// TIA Portal project "Shubra" (V16)

(* hardware
DEVICE "S7-1200 station_1"  S7-1200 Station
   slot 0: "Rack_0"  S7-1200 Rack  Rack  V1.0
   slot 1: "PLC_1"  CPU 1214C DC/DC/DC  6ES7 214-1AG40-0XB0  V4.4
   slot 2: "AI 8x13BIT_1"  6ES7 231-4HF32-0XB0  V2.1
DEVICE "PC-System_1"  SIMATIC PC station
   slot 0: "SIMATIC PC station"  Rail  SIMATIC PC-Station  V1.0
      slot 125: "Stationmanager"  Station_Manager  V6.0.4
   slot 1: "HMI_RT_1"  WinCC RT Advanced  6AV2 104-0xxxx-xxxx  16.0.0.0
      slot 33792: "Computer interface"  Host interface
   slot 2: "IE general_1"  IE General  IE_CP  V8.2.0
*)

// ===== PLC "PLC_1"  CPU 1214C DC/DC/DC =====

VAR_GLOBAL   // PLC tag table "Default tag table"
   "Tag_1" AT %IW112 : Int;
   "Tag_4" AT %IW114 : Int;
   "Tag_7" AT %IW116 : Int;
   "Tag_10" AT %IW118 : Int;
   "Tag_14" AT %IW120 : Int;
   "Tag_18" AT %IW122 : Int;
   "Tag_28" AT %IW124 : Int;
   "Tag_31" AT %IW126 : Int;
   "Tag_25" AT %I0.1 : Bool;
   "Tag_26" AT %I0.2 : Bool;
   "Tag_38" AT %I0.3 : Bool;
   "Axis_1_Pulse" AT %Q0.0 : Bool;
   "Axis_1_Direction" AT %Q0.1 : Bool;
   "Tag_17" AT %Q0.2 : Bool;
   "Axis_2_Pulse" AT %Q0.3 : Bool;
   "Axis_2_Direction" AT %Q0.4 : Bool;
   "Tag_22" AT %Q0.5 : Bool;
   "pump_run" AT %Q0.6 : Bool;
   "Tag_37" AT %QW128 : Word;
   "Tag_2" AT %MD40 : Real;
   "Suction_press" AT %MD44 : Real;
   "Tag_5" AT %MD48 : Real;
   "Discharge_Press" AT %MD52 : Real;
   "Tag_8" AT %MD56 : Real;
   "P3" AT %MD60 : Real;
   "Tag_12" AT %MD64 : Real;
   "P4" AT %MD68 : Real;
   "Tag_15" AT %MD72 : Real;
   "Temperature" AT %MD76 : Real;
   "Tag_20" AT %MD80 : Real;
   "Torque" AT %MD84 : Real;
   "Tag_29" AT %MD88 : Real;
   "RPM" AT %MD92 : Real;
   "Tag_32" AT %MD96 : Real;
   "vibration" AT %MD100 : Real;
   "Tag_11" AT %M20.0 : Bool;
   "compare" AT %MD104 : Real;
   "Tag_9" AT %M20.1 : Bool;
   "Tag_19" AT %M20.2 : Bool;
   "Tag_21" AT %M20.3 : Bool;
   "Tag_23" AT %M21.0 : Bool;
   "Tag_24" AT %M21.1 : Bool;
   "distance_1" AT %MD108 : Real;
   "Tag_35" AT %MD120 : Real;
   "Tag_36" AT %MD124 : DWord;
   "p3-p4" AT %MD128 : Real;
   "p3-p4_power5" AT %MD132 : Real;
   "p3-p4_power4" AT %MD136 : Real;
   "p3-p4_power3" AT %MD140 : Real;
   "p3-p4_power2" AT %MD144 : Real;
   "Q" AT %MD148 : Real;
   "VS" AT %MD152 : Real;
   "Vd" AT %MD156 : Real;
   "Vs2" AT %MD160 : Real;
   "Vd2" AT %MD164 : Real;
   "H" AT %MD168 : Real;
   "Shaft_power" AT %MD172 : Real;
   "Referance_motor_speed" AT %MD176 : Real;
   "QARS" AT %MD180 : Real;
   "Ref_speed_2" AT %MD184 : Real;
   "Ref_speed_3" AT %MD188 : Real;
   "motor_speed_2" AT %MD192 : Real;
   "motor_speed_3" AT %MD196 : Real;
   "H_ARS" AT %MD200 : Real;
   "SP_ARS" AT %MD204 : Real;
   "Efficiency" AT %MD208 : Real;
   "Npsh" AT %MD212 : Real;
   "Count_up" AT %M30.0 : Bool;
   "Tag_3" AT %M31.0 : Bool;
   "count_down" AT %M30.1 : Bool;
   "Tag_13" AT %M31.1 : Bool;
   "counter_reset" AT %M30.2 : Bool;
   "Tag_16" AT %MW36 : Int;
   "Raw1" AT %M30.3 : Bool;
   "raw2" AT %M30.4 : Bool;
   "raw3" AT %M30.5 : Bool;
   "raw4" AT %M30.6 : Bool;
   "raw5" AT %M30.7 : Bool;
   "raw6" AT %M31.4 : Bool;
   "record" AT %M31.5 : Bool;
   "stepp1_enab" AT %M31.6 : Bool;
   "stepp1_start" AT %M31.7 : Bool;
   "stepp1_distance" AT %MD216 : Real;
   "Tag_27" AT %M32.1 : Bool;
   "start_motor" AT %M32.2 : Bool;
   "clear All" AT %M32.3 : Bool;
   "open_close" AT %M32.4 : Bool;
   "stepp1_home" AT %M32.5 : Bool;
   "stepp2_home" AT %M32.6 : Bool;
   "stepp2_enab" AT %M32.7 : Bool;
   "stepp2_excut" AT %M33.0 : Bool;
   "stepp2_distance" AT %MD220 : Real;
   "Stepp1_dist_scale" AT %MD224 : Real;
   "Stepp2_dist_scale" AT %MD228 : Real;
   "configuration" AT %MW232 : WChar;
   "date" AT %MW234 : Date;
   "time" AT %MD236 : Time_Of_Day;
   "time_1" AT %MD240 : Time_Of_Day;
   "deviation" AT %MD244 : Real;
   "raw7" AT %M33.1 : Bool;
   "raw8" AT %M33.2 : Bool;
   "raw9" AT %M33.3 : Bool;
   "raw10" AT %M33.4 : Bool;
   "raw11" AT %M33.5 : Bool;
   "raw12" AT %M33.6 : Bool;
   "record1" AT %M33.7 : Bool;
   "Tag_6" AT %MD112 : Real;
END_VAR

DATA_BLOCK "P1P2"   // DB3
{ S7_Optimized_Access := 'TRUE' }
VERSION : 0.1
   VAR
      Pressurep1p2 : Array[0..23] of Real;
   END_VAR
BEGIN
END_DATA_BLOCK

DATA_BLOCK "P3P4"   // DB4
{ S7_Optimized_Access := 'TRUE' }
VERSION : 0.1
   VAR
      Pressure34 : Array[0..23] of Real;
   END_VAR
BEGIN
END_DATA_BLOCK

DATA_BLOCK "TS"   // DB5
{ S7_Optimized_Access := 'TRUE' }
VERSION : 0.1
   VAR
      TS : Array[0..23] of Real;
   END_VAR
BEGIN
END_DATA_BLOCK

DATA_BLOCK "Vib"   // DB6
{ S7_Optimized_Access := 'TRUE' }
VERSION : 0.1
   VAR
      vibration : Array[0..11] of Real;
   END_VAR
BEGIN
END_DATA_BLOCK

DATA_BLOCK "VSVD"   // DB7
{ S7_Optimized_Access := 'TRUE' }
VERSION : 0.1
   VAR
      VsVd : Array[0..23] of Real;
   END_VAR
BEGIN
END_DATA_BLOCK

DATA_BLOCK "QH"   // DB8
{ S7_Optimized_Access := 'TRUE' }
VERSION : 0.1
   VAR
      QH : Array[0..23] of Real;
   END_VAR
BEGIN
END_DATA_BLOCK

DATA_BLOCK "shftP.Pars"   // DB9
{ S7_Optimized_Access := 'TRUE' }
VERSION : 0.1
   VAR
      shaftP : Array[0..23] of Real;
   END_VAR
BEGIN
END_DATA_BLOCK

DATA_BLOCK "QarsHars"   // DB10
{ S7_Optimized_Access := 'TRUE' }
VERSION : 0.1
   VAR
      QarsHars : Array[0..23] of Real;
   END_VAR
BEGIN
END_DATA_BLOCK

DATA_BLOCK "EFF.NPSH"   // DB11
{ S7_Optimized_Access := 'TRUE' }
VERSION : 0.1
   VAR
      "EFF.NPSH" : Array[0..23] of Real;
   END_VAR
BEGIN
END_DATA_BLOCK

DATA_BLOCK "deviation_1"   // DB19
{ S7_Optimized_Access := 'TRUE' }
VERSION : 0.1
   VAR
      deviation : Real;
      deviation_1 : Real;
      deviation_2 : Real;
      deviation_3 : Real;
      deviation_4 : Real;
      deviation_5 : Real;
      deviation_0 : Real;
   END_VAR
BEGIN
END_DATA_BLOCK

// folder: System blocks/Program resources

DATA_BLOCK "IEC_Counter_0_DB"   // DB12
{ S7_Optimized_Access := 'TRUE' }
AUTHOR : Simatic
FAMILY : IEC
NAME : CNTR
VERSION : 1.0
// stored: InstanceOfName IEC_COUNTER
"IEC_COUNTER"
BEGIN
END_DATA_BLOCK

// folder: (top level)

DATA_BLOCK "Axis_1"   // DB1, Motion_DB
{ S7_Optimized_Access := 'TRUE' }
AUTHOR : SIMATIC
FAMILY : BasicMC
NAME : TO_PosAx
VERSION : 7.0
// stored: InstanceOfName TO_PositioningAxis
"TO_PositioningAxis"
BEGIN
   // Axis.OnlinePtoModeCU = 16#0000_0002
   // Axis.DirectionOutputEnabledCU = TRUE
   // Axis.SelectedChannel2EnumCU = %Q0.1
   // Axis.SelectedChannel1EnumCU = %Q0.0
   // Pulse.MinDeltaDeltaFrequencyCU = 0.004
   // Pulse.MaxDeltaDeltaFrequencyCU = 1.0E+10
   // Pulse.MinDeltaFrequencyCU = 0.005
   // Pulse.MaxDeltaFrequencyCU = 9.5E+9
   // Pulse.MinFrequencyCU = 1.0
   // Pulse.MaxFrequencyCU = 100000.0
   // Pulse.OutputSourceCU = 16#0000_0000
   // Axis.SelectPTO = 0
END_DATA_BLOCK

DATA_BLOCK "Axis_2"   // DB2, Motion_DB
{ S7_Optimized_Access := 'TRUE' }
AUTHOR : SIMATIC
FAMILY : BasicMC
NAME : TO_PosAx
VERSION : 7.0
// stored: InstanceOfName TO_PositioningAxis
"TO_PositioningAxis"
BEGIN
   // Axis.OnlinePtoModeCU = 16#0000_0002
   // Axis.DirectionOutputEnabledCU = TRUE
   // Axis.SelectedChannel2EnumCU = %Q0.4
   // Axis.SelectedChannel1EnumCU = %Q0.3
   // Pulse.MinDeltaDeltaFrequencyCU = 0.004
   // Pulse.MaxDeltaDeltaFrequencyCU = 1.0E+10
   // Pulse.MinDeltaFrequencyCU = 0.005
   // Pulse.MaxDeltaFrequencyCU = 9.5E+9
   // Pulse.MinFrequencyCU = 1.0
   // Pulse.MaxFrequencyCU = 100000.0
   // Pulse.OutputSourceCU = 16#0000_0000
   // Axis.SelectPTO = 1
   // Axis.OnlinePtoIndexCU = 1
END_DATA_BLOCK

FUNCTION "Analog input" : Void   // FC1, LAD
{ S7_Optimized_Access := 'TRUE' }
VERSION : 0.1
BEGIN

REGION Network 1: suction pressure
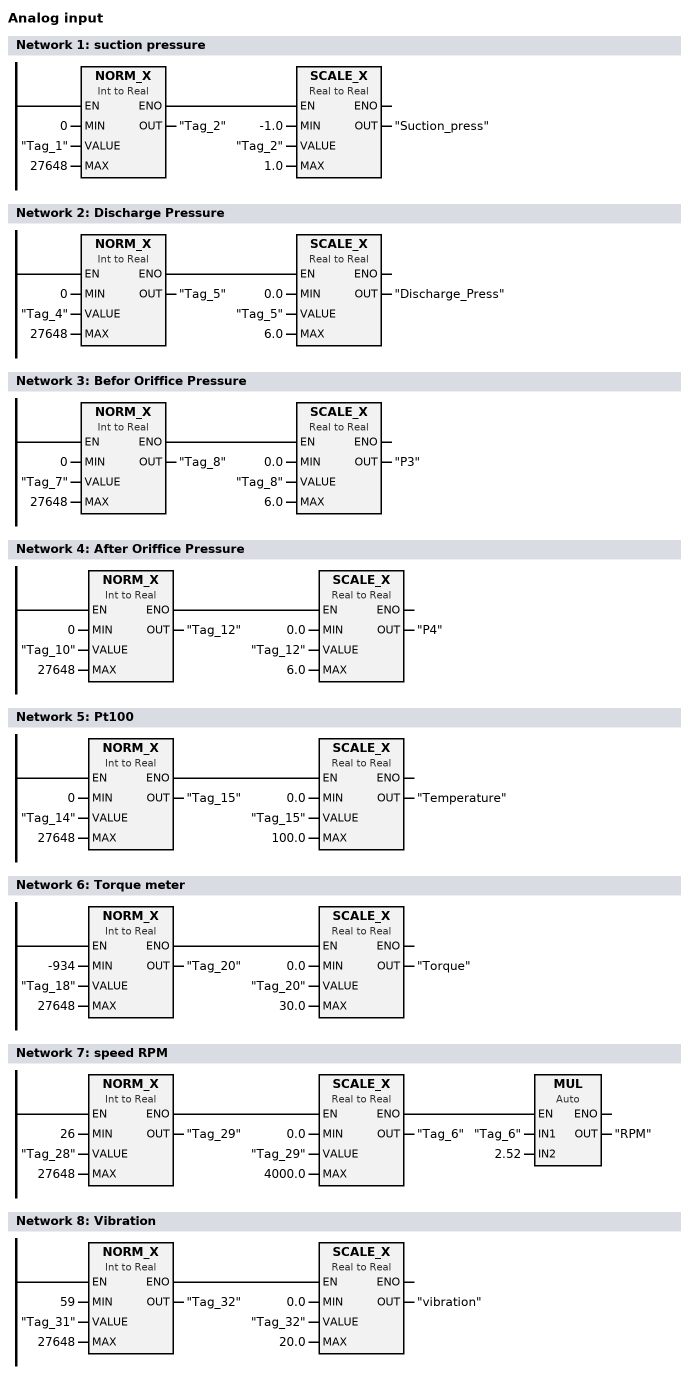
   RUNG wire#powerrail
      { S7_Templates := "[SrcType := Int, DestType := Real]" } Normalize(min := 0, value := "Tag_1", max := 27648, out => "Tag_2")
      { S7_Templates := "[SrcType := Real, DestType := Real]" } Scale(min := -1.0, value := "Tag_2", max := 1.0, out => "Suction_press")
   END_RUNG
   // the same network as SCL:
   "Tag_2" := NORM_X(MIN := 0, VALUE := "Tag_1", MAX := 27648);
   "Suction_press" := SCALE_X(MIN := -1.0, VALUE := "Tag_2", MAX := 1.0);
END_REGION

REGION Network 2: Discharge Pressure
   RUNG wire#powerrail
      { S7_Templates := "[SrcType := Int, DestType := Real]" } Normalize(min := 0, value := "Tag_4", max := 27648, out => "Tag_5")
      { S7_Templates := "[SrcType := Real, DestType := Real]" } Scale(min := 0.0, value := "Tag_5", max := 6.0, out => "Discharge_Press")
   END_RUNG
   // the same network as SCL:
   "Tag_5" := NORM_X(MIN := 0, VALUE := "Tag_4", MAX := 27648);
   "Discharge_Press" := SCALE_X(MIN := 0.0, VALUE := "Tag_5", MAX := 6.0);
END_REGION

REGION Network 3: Befor Oriffice Pressure
   RUNG wire#powerrail
      { S7_Templates := "[SrcType := Int, DestType := Real]" } Normalize(min := 0, value := "Tag_7", max := 27648, out => "Tag_8")
      { S7_Templates := "[SrcType := Real, DestType := Real]" } Scale(min := 0.0, value := "Tag_8", max := 6.0, out => "P3")
   END_RUNG
   // the same network as SCL:
   "Tag_8" := NORM_X(MIN := 0, VALUE := "Tag_7", MAX := 27648);
   "P3" := SCALE_X(MIN := 0.0, VALUE := "Tag_8", MAX := 6.0);
END_REGION

REGION Network 4: After Oriffice Pressure
   RUNG wire#powerrail
      { S7_Templates := "[SrcType := Int, DestType := Real]" } Normalize(min := 0, value := "Tag_10", max := 27648, out => "Tag_12")
      { S7_Templates := "[SrcType := Real, DestType := Real]" } Scale(min := 0.0, value := "Tag_12", max := 6.0, out => "P4")
   END_RUNG
   // the same network as SCL:
   "Tag_12" := NORM_X(MIN := 0, VALUE := "Tag_10", MAX := 27648);
   "P4" := SCALE_X(MIN := 0.0, VALUE := "Tag_12", MAX := 6.0);
END_REGION

REGION Network 5: Pt100
   RUNG wire#powerrail
      { S7_Templates := "[SrcType := Int, DestType := Real]" } Normalize(min := 0, value := "Tag_14", max := 27648, out => "Tag_15")
      { S7_Templates := "[SrcType := Real, DestType := Real]" } Scale(min := 0.0, value := "Tag_15", max := 100.0, out => "Temperature")
   END_RUNG
   // the same network as SCL:
   "Tag_15" := NORM_X(MIN := 0, VALUE := "Tag_14", MAX := 27648);
   "Temperature" := SCALE_X(MIN := 0.0, VALUE := "Tag_15", MAX := 100.0);
END_REGION

REGION Network 6: Torque meter
   RUNG wire#powerrail
      { S7_Templates := "[SrcType := Int, DestType := Real]" } Normalize(min := -934, value := "Tag_18", max := 27648, out => "Tag_20")
      { S7_Templates := "[SrcType := Real, DestType := Real]" } Scale(min := 0.0, value := "Tag_20", max := 30.0, out => "Torque")
   END_RUNG
   // the same network as SCL:
   "Tag_20" := NORM_X(MIN := -934, VALUE := "Tag_18", MAX := 27648);
   "Torque" := SCALE_X(MIN := 0.0, VALUE := "Tag_20", MAX := 30.0);
END_REGION

REGION Network 7: speed RPM
   RUNG wire#powerrail
      { S7_Templates := "[SrcType := Int, DestType := Real]" } Normalize(min := 26, value := "Tag_28", max := 27648, out => "Tag_29")
      { S7_Templates := "[SrcType := Real, DestType := Real]" } Scale(min := 0.0, value := "Tag_29", max := 4000.0, out => "Tag_6")
      Mul(in1 := "Tag_6", in2 := 2.52, out => "RPM")
   END_RUNG
   // the same network as SCL:
   "Tag_29" := NORM_X(MIN := 26, VALUE := "Tag_28", MAX := 27648);
   "Tag_6" := SCALE_X(MIN := 0.0, VALUE := "Tag_29", MAX := 4000.0);
   "RPM" := "Tag_6" * 2.52;
END_REGION

REGION Network 8: Vibration
   RUNG wire#powerrail
      { S7_Templates := "[SrcType := Int, DestType := Real]" } Normalize(min := 59, value := "Tag_31", max := 27648, out => "Tag_32")
      { S7_Templates := "[SrcType := Real, DestType := Real]" } Scale(min := 0.0, value := "Tag_32", max := 20.0, out => "vibration")
   END_RUNG
   // the same network as SCL:
   "Tag_32" := NORM_X(MIN := 59, VALUE := "Tag_31", MAX := 27648);
   "vibration" := SCALE_X(MIN := 0.0, VALUE := "Tag_32", MAX := 20.0);
END_REGION
END_FUNCTION

FUNCTION "clear_2" : Void   // FC2, LAD
{ S7_Optimized_Access := 'TRUE' }
VERSION : 0.1
BEGIN

REGION Network 2
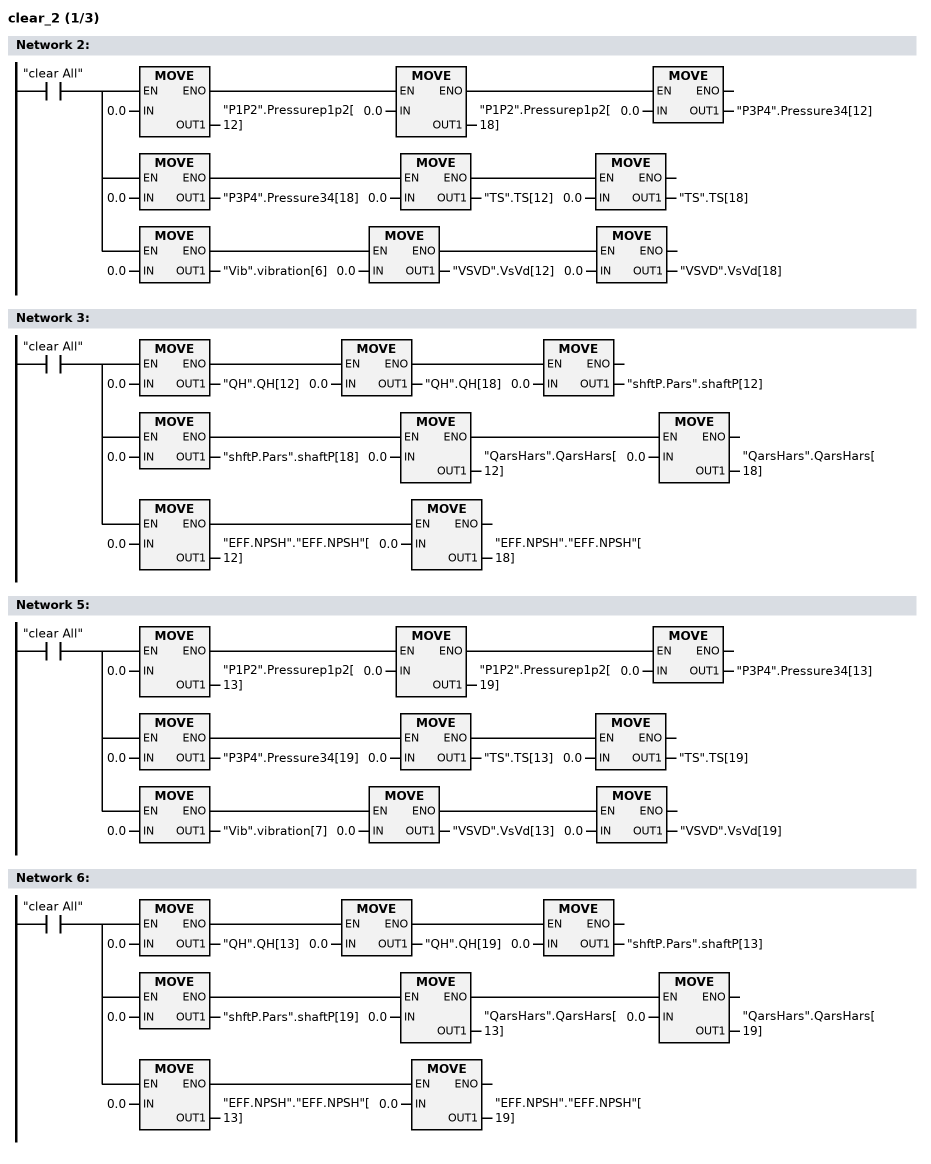
   RUNG wire#powerrail
      Contact( "clear All" )
      wire#w1
      Move(in := 0.0, out1 => "P1P2".Pressurep1p2[12])
      Move(in := 0.0, out1 => "P1P2".Pressurep1p2[18])
      Move(in := 0.0, out1 => "P3P4".Pressure34[12])
   END_RUNG
   RUNG wire#w1
      Move(in := 0.0, out1 => "P3P4".Pressure34[18])
      Move(in := 0.0, out1 => "TS".TS[12])
      Move(in := 0.0, out1 => "TS".TS[18])
   END_RUNG
   RUNG wire#w1
      Move(in := 0.0, out1 => "Vib".vibration[6])
      Move(in := 0.0, out1 => "VSVD".VsVd[12])
      Move(in := 0.0, out1 => "VSVD".VsVd[18])
   END_RUNG
   // the same network as SCL:
   IF "clear All" THEN
       "P1P2".Pressurep1p2[12] := 0.0;
       "P1P2".Pressurep1p2[18] := 0.0;
       "P3P4".Pressure34[12] := 0.0;
       "P3P4".Pressure34[18] := 0.0;
       "TS".TS[12] := 0.0;
       "TS".TS[18] := 0.0;
       "Vib".vibration[6] := 0.0;
       "VSVD".VsVd[12] := 0.0;
       "VSVD".VsVd[18] := 0.0;
   END_IF;
END_REGION

REGION Network 3
   RUNG wire#powerrail
      Contact( "clear All" )
      wire#w1
      Move(in := 0.0, out1 => "QH".QH[12])
      Move(in := 0.0, out1 => "QH".QH[18])
      Move(in := 0.0, out1 => "shftP.Pars".shaftP[12])
   END_RUNG
   RUNG wire#w1
      Move(in := 0.0, out1 => "shftP.Pars".shaftP[18])
      Move(in := 0.0, out1 => "QarsHars".QarsHars[12])
      Move(in := 0.0, out1 => "QarsHars".QarsHars[18])
   END_RUNG
   RUNG wire#w1
      Move(in := 0.0, out1 => "EFF.NPSH"."EFF.NPSH"[12])
      Move(in := 0.0, out1 => "EFF.NPSH"."EFF.NPSH"[18])
   END_RUNG
   // the same network as SCL:
   IF "clear All" THEN
       "QH".QH[12] := 0.0;
       "QH".QH[18] := 0.0;
       "shftP.Pars".shaftP[12] := 0.0;
       "shftP.Pars".shaftP[18] := 0.0;
       "QarsHars".QarsHars[12] := 0.0;
       "QarsHars".QarsHars[18] := 0.0;
       "EFF.NPSH"."EFF.NPSH"[12] := 0.0;
       "EFF.NPSH"."EFF.NPSH"[18] := 0.0;
   END_IF;
END_REGION

REGION Network 5
   RUNG wire#powerrail
      Contact( "clear All" )
      wire#w1
      Move(in := 0.0, out1 => "P1P2".Pressurep1p2[13])
      Move(in := 0.0, out1 => "P1P2".Pressurep1p2[19])
      Move(in := 0.0, out1 => "P3P4".Pressure34[13])
   END_RUNG
   RUNG wire#w1
      Move(in := 0.0, out1 => "P3P4".Pressure34[19])
      Move(in := 0.0, out1 => "TS".TS[13])
      Move(in := 0.0, out1 => "TS".TS[19])
   END_RUNG
   RUNG wire#w1
      Move(in := 0.0, out1 => "Vib".vibration[7])
      Move(in := 0.0, out1 => "VSVD".VsVd[13])
      Move(in := 0.0, out1 => "VSVD".VsVd[19])
   END_RUNG
   // the same network as SCL:
   IF "clear All" THEN
       "P1P2".Pressurep1p2[13] := 0.0;
       "P1P2".Pressurep1p2[19] := 0.0;
       "P3P4".Pressure34[13] := 0.0;
       "P3P4".Pressure34[19] := 0.0;
       "TS".TS[13] := 0.0;
       "TS".TS[19] := 0.0;
       "Vib".vibration[7] := 0.0;
       "VSVD".VsVd[13] := 0.0;
       "VSVD".VsVd[19] := 0.0;
   END_IF;
END_REGION

REGION Network 6
   RUNG wire#powerrail
      Contact( "clear All" )
      wire#w1
      Move(in := 0.0, out1 => "QH".QH[13])
      Move(in := 0.0, out1 => "QH".QH[19])
      Move(in := 0.0, out1 => "shftP.Pars".shaftP[13])
   END_RUNG
   RUNG wire#w1
      Move(in := 0.0, out1 => "shftP.Pars".shaftP[19])
      Move(in := 0.0, out1 => "QarsHars".QarsHars[13])
      Move(in := 0.0, out1 => "QarsHars".QarsHars[19])
   END_RUNG
   RUNG wire#w1
      Move(in := 0.0, out1 => "EFF.NPSH"."EFF.NPSH"[13])
      Move(in := 0.0, out1 => "EFF.NPSH"."EFF.NPSH"[19])
   END_RUNG
   // the same network as SCL:
   IF "clear All" THEN
       "QH".QH[13] := 0.0;
       "QH".QH[19] := 0.0;
       "shftP.Pars".shaftP[13] := 0.0;
       "shftP.Pars".shaftP[19] := 0.0;
       "QarsHars".QarsHars[13] := 0.0;
       "QarsHars".QarsHars[19] := 0.0;
       "EFF.NPSH"."EFF.NPSH"[13] := 0.0;
       "EFF.NPSH"."EFF.NPSH"[19] := 0.0;
   END_IF;
END_REGION

REGION Network 8
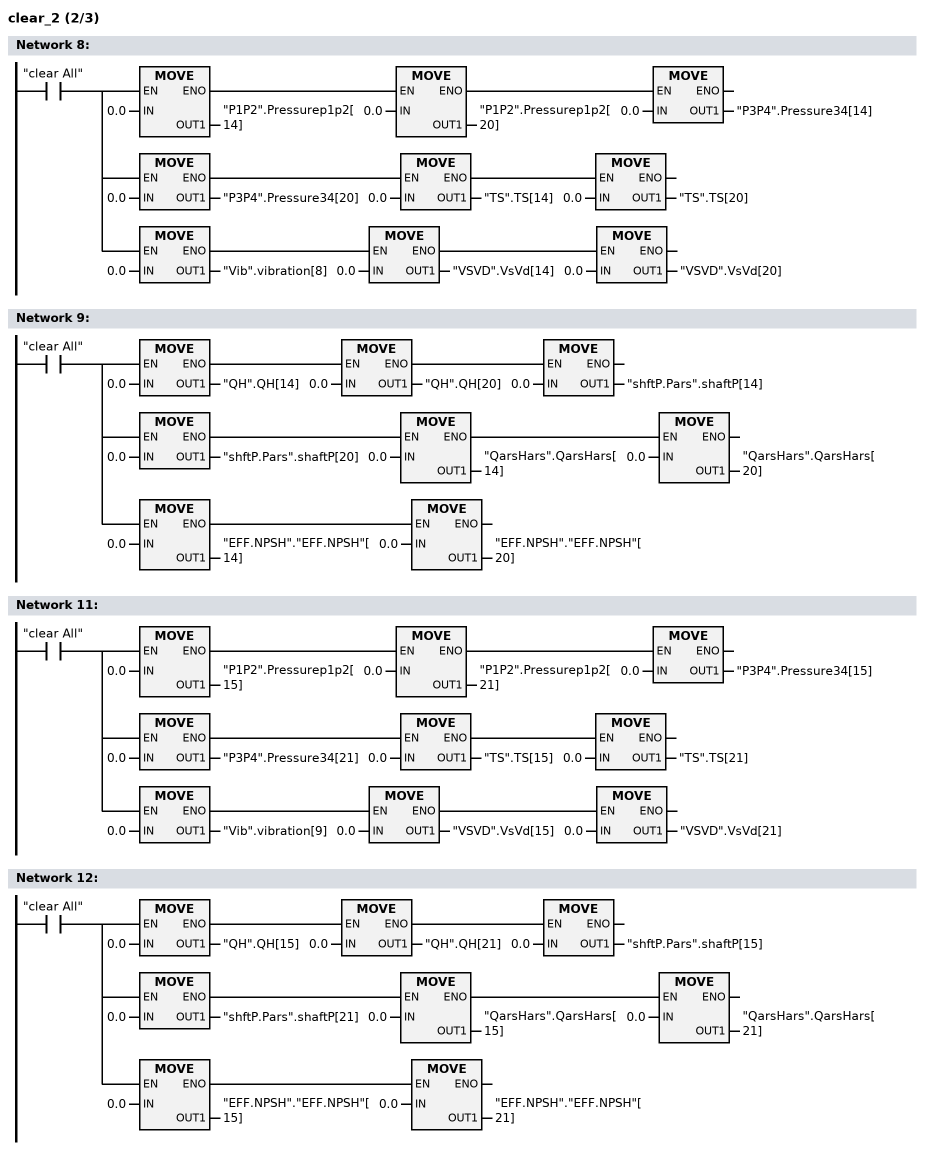
   RUNG wire#powerrail
      Contact( "clear All" )
      wire#w1
      Move(in := 0.0, out1 => "P1P2".Pressurep1p2[14])
      Move(in := 0.0, out1 => "P1P2".Pressurep1p2[20])
      Move(in := 0.0, out1 => "P3P4".Pressure34[14])
   END_RUNG
   RUNG wire#w1
      Move(in := 0.0, out1 => "P3P4".Pressure34[20])
      Move(in := 0.0, out1 => "TS".TS[14])
      Move(in := 0.0, out1 => "TS".TS[20])
   END_RUNG
   RUNG wire#w1
      Move(in := 0.0, out1 => "Vib".vibration[8])
      Move(in := 0.0, out1 => "VSVD".VsVd[14])
      Move(in := 0.0, out1 => "VSVD".VsVd[20])
   END_RUNG
   // the same network as SCL:
   IF "clear All" THEN
       "P1P2".Pressurep1p2[14] := 0.0;
       "P1P2".Pressurep1p2[20] := 0.0;
       "P3P4".Pressure34[14] := 0.0;
       "P3P4".Pressure34[20] := 0.0;
       "TS".TS[14] := 0.0;
       "TS".TS[20] := 0.0;
       "Vib".vibration[8] := 0.0;
       "VSVD".VsVd[14] := 0.0;
       "VSVD".VsVd[20] := 0.0;
   END_IF;
END_REGION

REGION Network 9
   RUNG wire#powerrail
      Contact( "clear All" )
      wire#w1
      Move(in := 0.0, out1 => "QH".QH[14])
      Move(in := 0.0, out1 => "QH".QH[20])
      Move(in := 0.0, out1 => "shftP.Pars".shaftP[14])
   END_RUNG
   RUNG wire#w1
      Move(in := 0.0, out1 => "shftP.Pars".shaftP[20])
      Move(in := 0.0, out1 => "QarsHars".QarsHars[14])
      Move(in := 0.0, out1 => "QarsHars".QarsHars[20])
   END_RUNG
   RUNG wire#w1
      Move(in := 0.0, out1 => "EFF.NPSH"."EFF.NPSH"[14])
      Move(in := 0.0, out1 => "EFF.NPSH"."EFF.NPSH"[20])
   END_RUNG
   // the same network as SCL:
   IF "clear All" THEN
       "QH".QH[14] := 0.0;
       "QH".QH[20] := 0.0;
       "shftP.Pars".shaftP[14] := 0.0;
       "shftP.Pars".shaftP[20] := 0.0;
       "QarsHars".QarsHars[14] := 0.0;
       "QarsHars".QarsHars[20] := 0.0;
       "EFF.NPSH"."EFF.NPSH"[14] := 0.0;
       "EFF.NPSH"."EFF.NPSH"[20] := 0.0;
   END_IF;
END_REGION

REGION Network 11
   RUNG wire#powerrail
      Contact( "clear All" )
      wire#w1
      Move(in := 0.0, out1 => "P1P2".Pressurep1p2[15])
      Move(in := 0.0, out1 => "P1P2".Pressurep1p2[21])
      Move(in := 0.0, out1 => "P3P4".Pressure34[15])
   END_RUNG
   RUNG wire#w1
      Move(in := 0.0, out1 => "P3P4".Pressure34[21])
      Move(in := 0.0, out1 => "TS".TS[15])
      Move(in := 0.0, out1 => "TS".TS[21])
   END_RUNG
   RUNG wire#w1
      Move(in := 0.0, out1 => "Vib".vibration[9])
      Move(in := 0.0, out1 => "VSVD".VsVd[15])
      Move(in := 0.0, out1 => "VSVD".VsVd[21])
   END_RUNG
   // the same network as SCL:
   IF "clear All" THEN
       "P1P2".Pressurep1p2[15] := 0.0;
       "P1P2".Pressurep1p2[21] := 0.0;
       "P3P4".Pressure34[15] := 0.0;
       "P3P4".Pressure34[21] := 0.0;
       "TS".TS[15] := 0.0;
       "TS".TS[21] := 0.0;
       "Vib".vibration[9] := 0.0;
       "VSVD".VsVd[15] := 0.0;
       "VSVD".VsVd[21] := 0.0;
   END_IF;
END_REGION

REGION Network 12
   RUNG wire#powerrail
      Contact( "clear All" )
      wire#w1
      Move(in := 0.0, out1 => "QH".QH[15])
      Move(in := 0.0, out1 => "QH".QH[21])
      Move(in := 0.0, out1 => "shftP.Pars".shaftP[15])
   END_RUNG
   RUNG wire#w1
      Move(in := 0.0, out1 => "shftP.Pars".shaftP[21])
      Move(in := 0.0, out1 => "QarsHars".QarsHars[15])
      Move(in := 0.0, out1 => "QarsHars".QarsHars[21])
   END_RUNG
   RUNG wire#w1
      Move(in := 0.0, out1 => "EFF.NPSH"."EFF.NPSH"[15])
      Move(in := 0.0, out1 => "EFF.NPSH"."EFF.NPSH"[21])
   END_RUNG
   // the same network as SCL:
   IF "clear All" THEN
       "QH".QH[15] := 0.0;
       "QH".QH[21] := 0.0;
       "shftP.Pars".shaftP[15] := 0.0;
       "shftP.Pars".shaftP[21] := 0.0;
       "QarsHars".QarsHars[15] := 0.0;
       "QarsHars".QarsHars[21] := 0.0;
       "EFF.NPSH"."EFF.NPSH"[15] := 0.0;
       "EFF.NPSH"."EFF.NPSH"[21] := 0.0;
   END_IF;
END_REGION

REGION Network 14
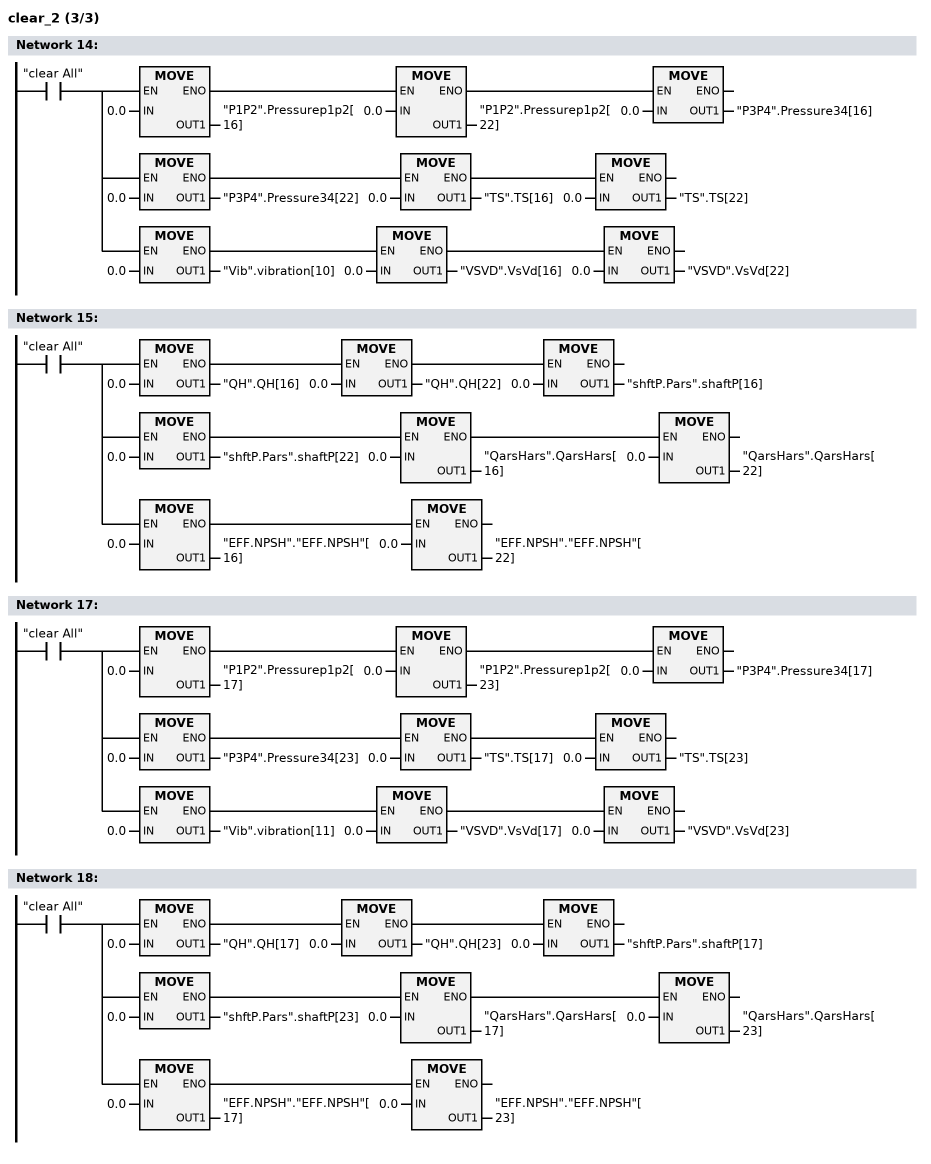
   RUNG wire#powerrail
      Contact( "clear All" )
      wire#w1
      Move(in := 0.0, out1 => "P1P2".Pressurep1p2[16])
      Move(in := 0.0, out1 => "P1P2".Pressurep1p2[22])
      Move(in := 0.0, out1 => "P3P4".Pressure34[16])
   END_RUNG
   RUNG wire#w1
      Move(in := 0.0, out1 => "P3P4".Pressure34[22])
      Move(in := 0.0, out1 => "TS".TS[16])
      Move(in := 0.0, out1 => "TS".TS[22])
   END_RUNG
   RUNG wire#w1
      Move(in := 0.0, out1 => "Vib".vibration[10])
      Move(in := 0.0, out1 => "VSVD".VsVd[16])
      Move(in := 0.0, out1 => "VSVD".VsVd[22])
   END_RUNG
   // the same network as SCL:
   IF "clear All" THEN
       "P1P2".Pressurep1p2[16] := 0.0;
       "P1P2".Pressurep1p2[22] := 0.0;
       "P3P4".Pressure34[16] := 0.0;
       "P3P4".Pressure34[22] := 0.0;
       "TS".TS[16] := 0.0;
       "TS".TS[22] := 0.0;
       "Vib".vibration[10] := 0.0;
       "VSVD".VsVd[16] := 0.0;
       "VSVD".VsVd[22] := 0.0;
   END_IF;
END_REGION

REGION Network 15
   RUNG wire#powerrail
      Contact( "clear All" )
      wire#w1
      Move(in := 0.0, out1 => "QH".QH[16])
      Move(in := 0.0, out1 => "QH".QH[22])
      Move(in := 0.0, out1 => "shftP.Pars".shaftP[16])
   END_RUNG
   RUNG wire#w1
      Move(in := 0.0, out1 => "shftP.Pars".shaftP[22])
      Move(in := 0.0, out1 => "QarsHars".QarsHars[16])
      Move(in := 0.0, out1 => "QarsHars".QarsHars[22])
   END_RUNG
   RUNG wire#w1
      Move(in := 0.0, out1 => "EFF.NPSH"."EFF.NPSH"[16])
      Move(in := 0.0, out1 => "EFF.NPSH"."EFF.NPSH"[22])
   END_RUNG
   // the same network as SCL:
   IF "clear All" THEN
       "QH".QH[16] := 0.0;
       "QH".QH[22] := 0.0;
       "shftP.Pars".shaftP[16] := 0.0;
       "shftP.Pars".shaftP[22] := 0.0;
       "QarsHars".QarsHars[16] := 0.0;
       "QarsHars".QarsHars[22] := 0.0;
       "EFF.NPSH"."EFF.NPSH"[16] := 0.0;
       "EFF.NPSH"."EFF.NPSH"[22] := 0.0;
   END_IF;
END_REGION

REGION Network 17
   RUNG wire#powerrail
      Contact( "clear All" )
      wire#w1
      Move(in := 0.0, out1 => "P1P2".Pressurep1p2[17])
      Move(in := 0.0, out1 => "P1P2".Pressurep1p2[23])
      Move(in := 0.0, out1 => "P3P4".Pressure34[17])
   END_RUNG
   RUNG wire#w1
      Move(in := 0.0, out1 => "P3P4".Pressure34[23])
      Move(in := 0.0, out1 => "TS".TS[17])
      Move(in := 0.0, out1 => "TS".TS[23])
   END_RUNG
   RUNG wire#w1
      Move(in := 0.0, out1 => "Vib".vibration[11])
      Move(in := 0.0, out1 => "VSVD".VsVd[17])
      Move(in := 0.0, out1 => "VSVD".VsVd[23])
   END_RUNG
   // the same network as SCL:
   IF "clear All" THEN
       "P1P2".Pressurep1p2[17] := 0.0;
       "P1P2".Pressurep1p2[23] := 0.0;
       "P3P4".Pressure34[17] := 0.0;
       "P3P4".Pressure34[23] := 0.0;
       "TS".TS[17] := 0.0;
       "TS".TS[23] := 0.0;
       "Vib".vibration[11] := 0.0;
       "VSVD".VsVd[17] := 0.0;
       "VSVD".VsVd[23] := 0.0;
   END_IF;
END_REGION

REGION Network 18
   RUNG wire#powerrail
      Contact( "clear All" )
      wire#w1
      Move(in := 0.0, out1 => "QH".QH[17])
      Move(in := 0.0, out1 => "QH".QH[23])
      Move(in := 0.0, out1 => "shftP.Pars".shaftP[17])
   END_RUNG
   RUNG wire#w1
      Move(in := 0.0, out1 => "shftP.Pars".shaftP[23])
      Move(in := 0.0, out1 => "QarsHars".QarsHars[17])
      Move(in := 0.0, out1 => "QarsHars".QarsHars[23])
   END_RUNG
   RUNG wire#w1
      Move(in := 0.0, out1 => "EFF.NPSH"."EFF.NPSH"[17])
      Move(in := 0.0, out1 => "EFF.NPSH"."EFF.NPSH"[23])
   END_RUNG
   // the same network as SCL:
   IF "clear All" THEN
       "QH".QH[17] := 0.0;
       "QH".QH[23] := 0.0;
       "shftP.Pars".shaftP[17] := 0.0;
       "shftP.Pars".shaftP[23] := 0.0;
       "QarsHars".QarsHars[17] := 0.0;
       "QarsHars".QarsHars[23] := 0.0;
       "EFF.NPSH"."EFF.NPSH"[17] := 0.0;
       "EFF.NPSH"."EFF.NPSH"[23] := 0.0;
   END_IF;
END_REGION
END_FUNCTION

FUNCTION "calculation" : Void   // FC3, LAD
{ S7_Optimized_Access := 'TRUE' }
VERSION : 0.1
BEGIN

REGION Network 1
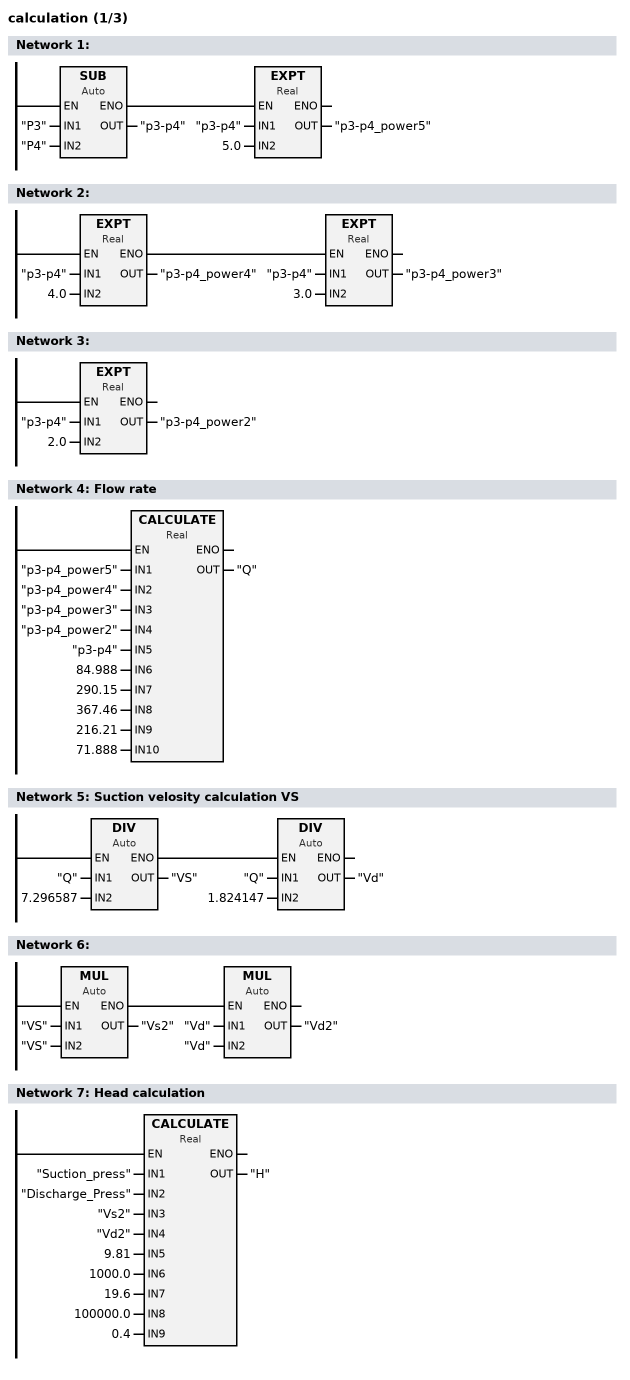
   "p3-p4" := "P3" - "P4";
   "p3-p4_power5" := "p3-p4" ** 5.0;
END_REGION

REGION Network 2
   "p3-p4_power4" := "p3-p4" ** 4.0;
   "p3-p4_power3" := "p3-p4" ** 3.0;
END_REGION

REGION Network 3
   "p3-p4_power2" := "p3-p4" ** 2.0;
END_REGION

REGION Network 4: Flow rate
   RUNG wire#powerrail
      { S7_Templates := "SrcType := Real"; S7_Expression := "(IN1*IN6)-(IN2*IN7)+(IN3*IN8)-(IN4*IN9)+(IN5*IN10)" } Calculate(in1 := "p3-p4_power5", in2 := "p3-p4_power4", in3 := "p3-p4_power3", in4 := "p3-p4_power2", in5 := "p3-p4", in6 := 84.988, in7 := 290.15, in8 := 367.46, in9 := 216.21, in10 := 71.888, out => "Q")
   END_RUNG
   // the same network as SCL:
   "Q" := ("p3-p4_power5"*84.988)-("p3-p4_power4"*290.15)+("p3-p4_power3"*367.46)-("p3-p4_power2"*216.21)+("p3-p4"*71.888);
END_REGION

REGION Network 5: Suction velosity calculation VS
   RUNG wire#powerrail
      Div(in1 := "Q", in2 := 7.296587, out => "VS")
      Div(in1 := "Q", in2 := 1.824147, out => "Vd")
   END_RUNG
   // the same network as SCL:
   "VS" := "Q" / 7.296587;
   "Vd" := "Q" / 1.824147;
END_REGION

REGION Network 6
   RUNG wire#powerrail
      Mul(in1 := "VS", in2 := "VS", out => "Vs2")
      Mul(in1 := "Vd", in2 := "Vd", out => "Vd2")
   END_RUNG
   // the same network as SCL:
   "Vs2" := "VS" * "VS";
   "Vd2" := "Vd" * "Vd";
END_REGION

REGION Network 7: Head calculation
   RUNG wire#powerrail
      { S7_Templates := "SrcType := Real"; S7_Expression := "(((IN2-IN1)/(IN5*IN6))*IN8)+((IN4-IN3)/IN7)+IN9" } Calculate(in1 := "Suction_press", in2 := "Discharge_Press", in3 := "Vs2", in4 := "Vd2", in5 := 9.81, in6 := 1000.0, in7 := 19.6, in8 := 100000.0, in9 := 0.4, out => "H")
   END_RUNG
   // the same network as SCL:
   "H" := ((("Discharge_Press"-"Suction_press")/(9.81*1000.0))*100000.0)+(("Vd2"-"Vs2")/19.6)+0.4;
END_REGION

REGION Network 8: Shaft power calculation
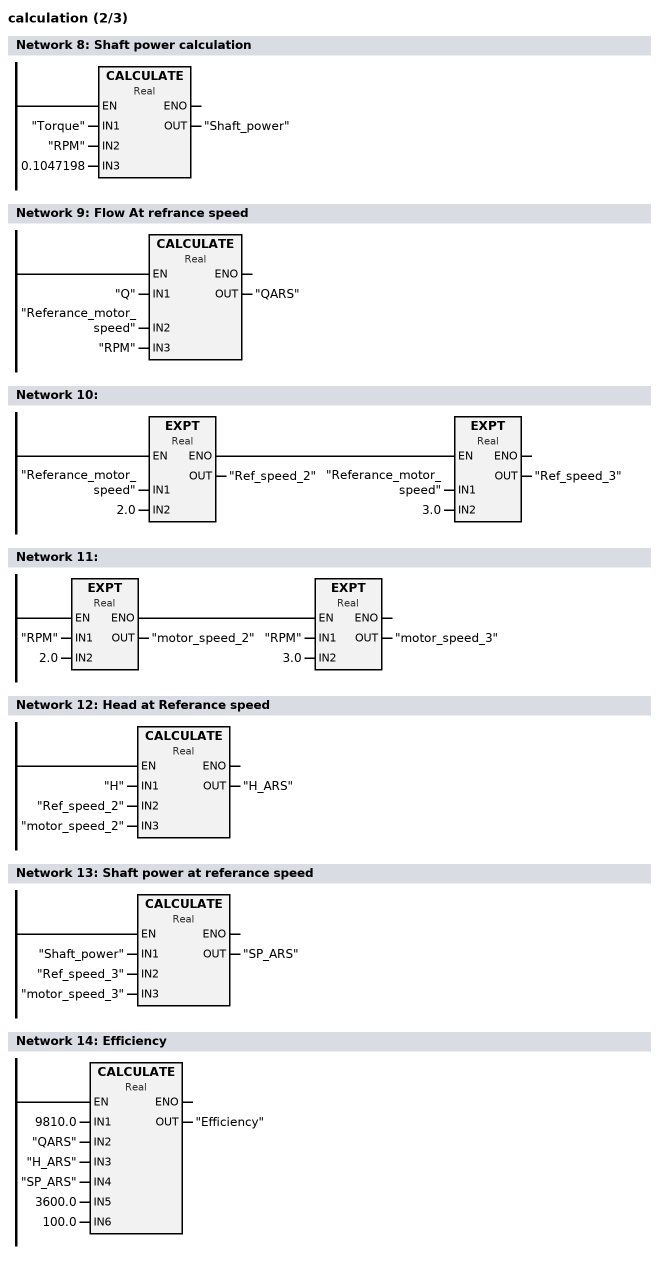
   RUNG wire#powerrail
      { S7_Templates := "SrcType := Real"; S7_Expression := "IN1*IN2*IN3" } Calculate(in1 := "Torque", in2 := "RPM", in3 := 0.1047198, out => "Shaft_power")
   END_RUNG
   // the same network as SCL:
   "Shaft_power" := "Torque"*"RPM"*0.1047198;
END_REGION

REGION Network 9: Flow At refrance speed
   RUNG wire#powerrail
      { S7_Templates := "SrcType := Real"; S7_Expression := "IN1*(IN2/IN3)" } Calculate(in1 := "Q", in2 := "Referance_motor_speed", in3 := "RPM", out => "QARS")
   END_RUNG
   // the same network as SCL:
   "QARS" := "Q"*("Referance_motor_speed"/"RPM");
END_REGION

REGION Network 10
   "Ref_speed_2" := "Referance_motor_speed" ** 2.0;
   "Ref_speed_3" := "Referance_motor_speed" ** 3.0;
END_REGION

REGION Network 11
   "motor_speed_2" := "RPM" ** 2.0;
   "motor_speed_3" := "RPM" ** 3.0;
END_REGION

REGION Network 12: Head at Referance speed
   RUNG wire#powerrail
      { S7_Templates := "SrcType := Real"; S7_Expression := "IN1*(IN2/IN3)" } Calculate(in1 := "H", in2 := "Ref_speed_2", in3 := "motor_speed_2", out => "H_ARS")
   END_RUNG
   // the same network as SCL:
   "H_ARS" := "H"*("Ref_speed_2"/"motor_speed_2");
END_REGION

REGION Network 13: Shaft power at referance speed
   RUNG wire#powerrail
      { S7_Templates := "SrcType := Real"; S7_Expression := "IN1*(IN2/IN3)" } Calculate(in1 := "Shaft_power", in2 := "Ref_speed_3", in3 := "motor_speed_3", out => "SP_ARS")
   END_RUNG
   // the same network as SCL:
   "SP_ARS" := "Shaft_power"*("Ref_speed_3"/"motor_speed_3");
END_REGION

REGION Network 14: Efficiency
   RUNG wire#powerrail
      { S7_Templates := "SrcType := Real"; S7_Expression := "((IN1*IN2*IN3)/(IN4*IN5))*IN6" } Calculate(in1 := 9810.0, in2 := "QARS", in3 := "H_ARS", in4 := "SP_ARS", in5 := 3600.0, in6 := 100.0, out => "Efficiency")
   END_RUNG
   // the same network as SCL:
   "Efficiency" := ((9810.0*"QARS"*"H_ARS")/("SP_ARS"*3600.0))*100.0;
END_REGION

REGION Network 15
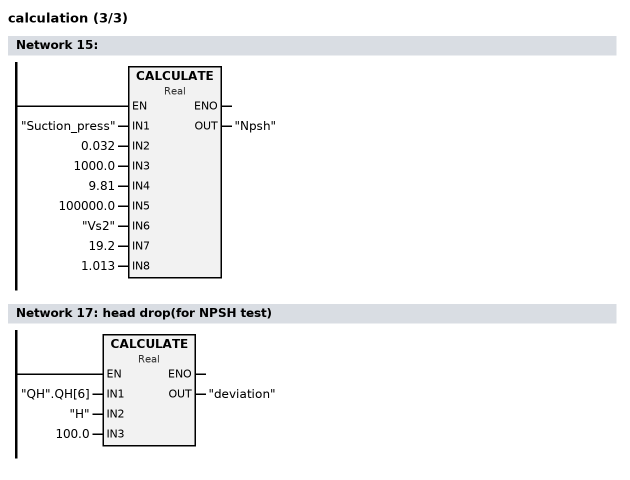
   RUNG wire#powerrail
      { S7_Templates := "SrcType := Real"; S7_Expression := "(((IN1-IN2)/(IN3*IN4))*IN5)+(IN6/IN7)+((IN8*IN5)/(IN3*IN4))" } Calculate(in1 := "Suction_press", in2 := 0.032, in3 := 1000.0, in4 := 9.81, in5 := 100000.0, in6 := "Vs2", in7 := 19.2, in8 := 1.013, out => "Npsh")
   END_RUNG
   // the same network as SCL:
   "Npsh" := ((("Suction_press"-0.032)/(1000.0*9.81))*100000.0)+("Vs2"/19.2)+((1.013*100000.0)/(1000.0*9.81));
END_REGION

REGION Network 17: head drop(for NPSH test)
   RUNG wire#powerrail
      { S7_Templates := "SrcType := Real"; S7_Expression := "((IN1-IN2)/IN1)*IN3" } Calculate(in1 := "QH".QH[6], in2 := "H", in3 := 100.0, out => "deviation")
   END_RUNG
   // the same network as SCL:
   "deviation" := (("QH".QH[6]-"H")/"QH".QH[6])*100.0;
END_REGION
END_FUNCTION

FUNCTION "move" : Void   // FC4, LAD
{ S7_Optimized_Access := 'TRUE' }
VERSION : 0.1
BEGIN

REGION Network 2
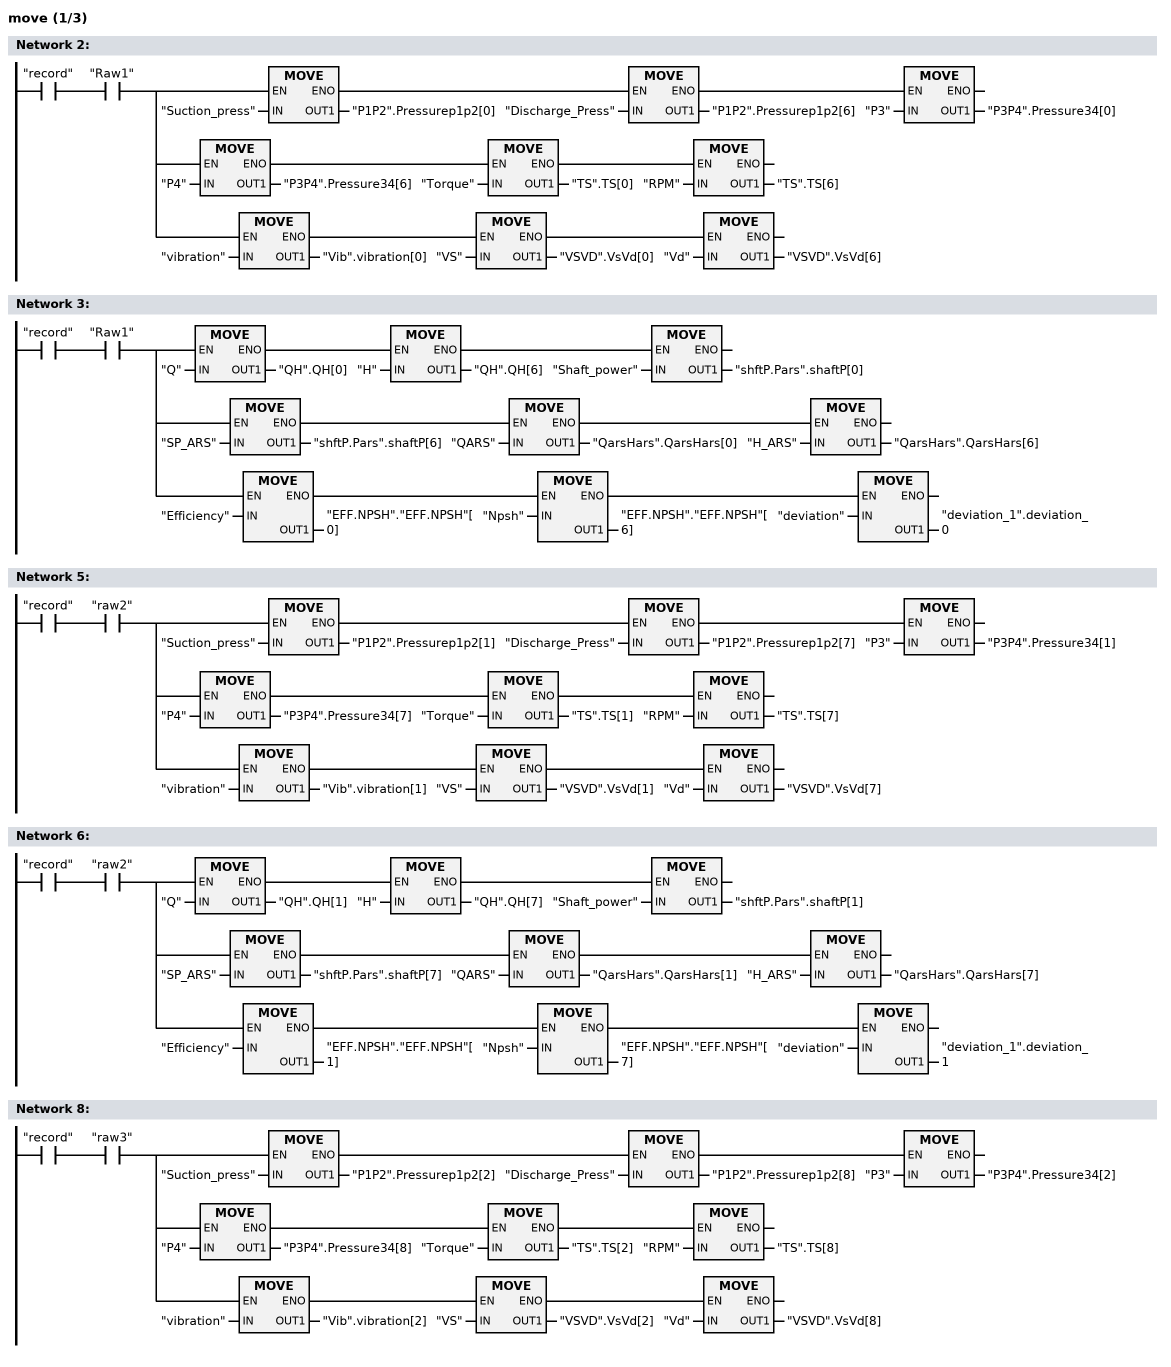
   RUNG wire#powerrail
      Contact( "record" )
      Contact( "Raw1" )
      wire#w1
      Move(in := "Suction_press", out1 => "P1P2".Pressurep1p2[0])
      Move(in := "Discharge_Press", out1 => "P1P2".Pressurep1p2[6])
      Move(in := "P3", out1 => "P3P4".Pressure34[0])
   END_RUNG
   RUNG wire#w1
      Move(in := "P4", out1 => "P3P4".Pressure34[6])
      Move(in := "Torque", out1 => "TS".TS[0])
      Move(in := "RPM", out1 => "TS".TS[6])
   END_RUNG
   RUNG wire#w1
      Move(in := "vibration", out1 => "Vib".vibration[0])
      Move(in := "VS", out1 => "VSVD".VsVd[0])
      Move(in := "Vd", out1 => "VSVD".VsVd[6])
   END_RUNG
   // the same network as SCL:
   IF "record" AND "Raw1" THEN
       "P1P2".Pressurep1p2[0] := "Suction_press";
       "P1P2".Pressurep1p2[6] := "Discharge_Press";
       "P3P4".Pressure34[0] := "P3";
       "P3P4".Pressure34[6] := "P4";
       "TS".TS[0] := "Torque";
       "TS".TS[6] := "RPM";
       "Vib".vibration[0] := "vibration";
       "VSVD".VsVd[0] := "VS";
       "VSVD".VsVd[6] := "Vd";
   END_IF;
END_REGION

REGION Network 3
   RUNG wire#powerrail
      Contact( "record" )
      Contact( "Raw1" )
      wire#w1
      Move(in := "Q", out1 => "QH".QH[0])
      Move(in := "H", out1 => "QH".QH[6])
      Move(in := "Shaft_power", out1 => "shftP.Pars".shaftP[0])
   END_RUNG
   RUNG wire#w1
      Move(in := "SP_ARS", out1 => "shftP.Pars".shaftP[6])
      Move(in := "QARS", out1 => "QarsHars".QarsHars[0])
      Move(in := "H_ARS", out1 => "QarsHars".QarsHars[6])
   END_RUNG
   RUNG wire#w1
      Move(in := "Efficiency", out1 => "EFF.NPSH"."EFF.NPSH"[0])
      Move(in := "Npsh", out1 => "EFF.NPSH"."EFF.NPSH"[6])
      Move(in := "deviation", out1 => "deviation_1".deviation_0)
   END_RUNG
   // the same network as SCL:
   IF "record" AND "Raw1" THEN
       "QH".QH[0] := "Q";
       "QH".QH[6] := "H";
       "shftP.Pars".shaftP[0] := "Shaft_power";
       "shftP.Pars".shaftP[6] := "SP_ARS";
       "QarsHars".QarsHars[0] := "QARS";
       "QarsHars".QarsHars[6] := "H_ARS";
       "EFF.NPSH"."EFF.NPSH"[0] := "Efficiency";
       "EFF.NPSH"."EFF.NPSH"[6] := "Npsh";
       "deviation_1".deviation_0 := "deviation";
   END_IF;
END_REGION

REGION Network 5
   RUNG wire#powerrail
      Contact( "record" )
      Contact( "raw2" )
      wire#w1
      Move(in := "Suction_press", out1 => "P1P2".Pressurep1p2[1])
      Move(in := "Discharge_Press", out1 => "P1P2".Pressurep1p2[7])
      Move(in := "P3", out1 => "P3P4".Pressure34[1])
   END_RUNG
   RUNG wire#w1
      Move(in := "P4", out1 => "P3P4".Pressure34[7])
      Move(in := "Torque", out1 => "TS".TS[1])
      Move(in := "RPM", out1 => "TS".TS[7])
   END_RUNG
   RUNG wire#w1
      Move(in := "vibration", out1 => "Vib".vibration[1])
      Move(in := "VS", out1 => "VSVD".VsVd[1])
      Move(in := "Vd", out1 => "VSVD".VsVd[7])
   END_RUNG
   // the same network as SCL:
   IF "record" AND "raw2" THEN
       "P1P2".Pressurep1p2[1] := "Suction_press";
       "P1P2".Pressurep1p2[7] := "Discharge_Press";
       "P3P4".Pressure34[1] := "P3";
       "P3P4".Pressure34[7] := "P4";
       "TS".TS[1] := "Torque";
       "TS".TS[7] := "RPM";
       "Vib".vibration[1] := "vibration";
       "VSVD".VsVd[1] := "VS";
       "VSVD".VsVd[7] := "Vd";
   END_IF;
END_REGION

REGION Network 6
   RUNG wire#powerrail
      Contact( "record" )
      Contact( "raw2" )
      wire#w1
      Move(in := "Q", out1 => "QH".QH[1])
      Move(in := "H", out1 => "QH".QH[7])
      Move(in := "Shaft_power", out1 => "shftP.Pars".shaftP[1])
   END_RUNG
   RUNG wire#w1
      Move(in := "SP_ARS", out1 => "shftP.Pars".shaftP[7])
      Move(in := "QARS", out1 => "QarsHars".QarsHars[1])
      Move(in := "H_ARS", out1 => "QarsHars".QarsHars[7])
   END_RUNG
   RUNG wire#w1
      Move(in := "Efficiency", out1 => "EFF.NPSH"."EFF.NPSH"[1])
      Move(in := "Npsh", out1 => "EFF.NPSH"."EFF.NPSH"[7])
      Move(in := "deviation", out1 => "deviation_1".deviation_1)
   END_RUNG
   // the same network as SCL:
   IF "record" AND "raw2" THEN
       "QH".QH[1] := "Q";
       "QH".QH[7] := "H";
       "shftP.Pars".shaftP[1] := "Shaft_power";
       "shftP.Pars".shaftP[7] := "SP_ARS";
       "QarsHars".QarsHars[1] := "QARS";
       "QarsHars".QarsHars[7] := "H_ARS";
       "EFF.NPSH"."EFF.NPSH"[1] := "Efficiency";
       "EFF.NPSH"."EFF.NPSH"[7] := "Npsh";
       "deviation_1".deviation_1 := "deviation";
   END_IF;
END_REGION

REGION Network 8
   RUNG wire#powerrail
      Contact( "record" )
      Contact( "raw3" )
      wire#w1
      Move(in := "Suction_press", out1 => "P1P2".Pressurep1p2[2])
      Move(in := "Discharge_Press", out1 => "P1P2".Pressurep1p2[8])
      Move(in := "P3", out1 => "P3P4".Pressure34[2])
   END_RUNG
   RUNG wire#w1
      Move(in := "P4", out1 => "P3P4".Pressure34[8])
      Move(in := "Torque", out1 => "TS".TS[2])
      Move(in := "RPM", out1 => "TS".TS[8])
   END_RUNG
   RUNG wire#w1
      Move(in := "vibration", out1 => "Vib".vibration[2])
      Move(in := "VS", out1 => "VSVD".VsVd[2])
      Move(in := "Vd", out1 => "VSVD".VsVd[8])
   END_RUNG
   // the same network as SCL:
   IF "record" AND "raw3" THEN
       "P1P2".Pressurep1p2[2] := "Suction_press";
       "P1P2".Pressurep1p2[8] := "Discharge_Press";
       "P3P4".Pressure34[2] := "P3";
       "P3P4".Pressure34[8] := "P4";
       "TS".TS[2] := "Torque";
       "TS".TS[8] := "RPM";
       "Vib".vibration[2] := "vibration";
       "VSVD".VsVd[2] := "VS";
       "VSVD".VsVd[8] := "Vd";
   END_IF;
END_REGION

REGION Network 9
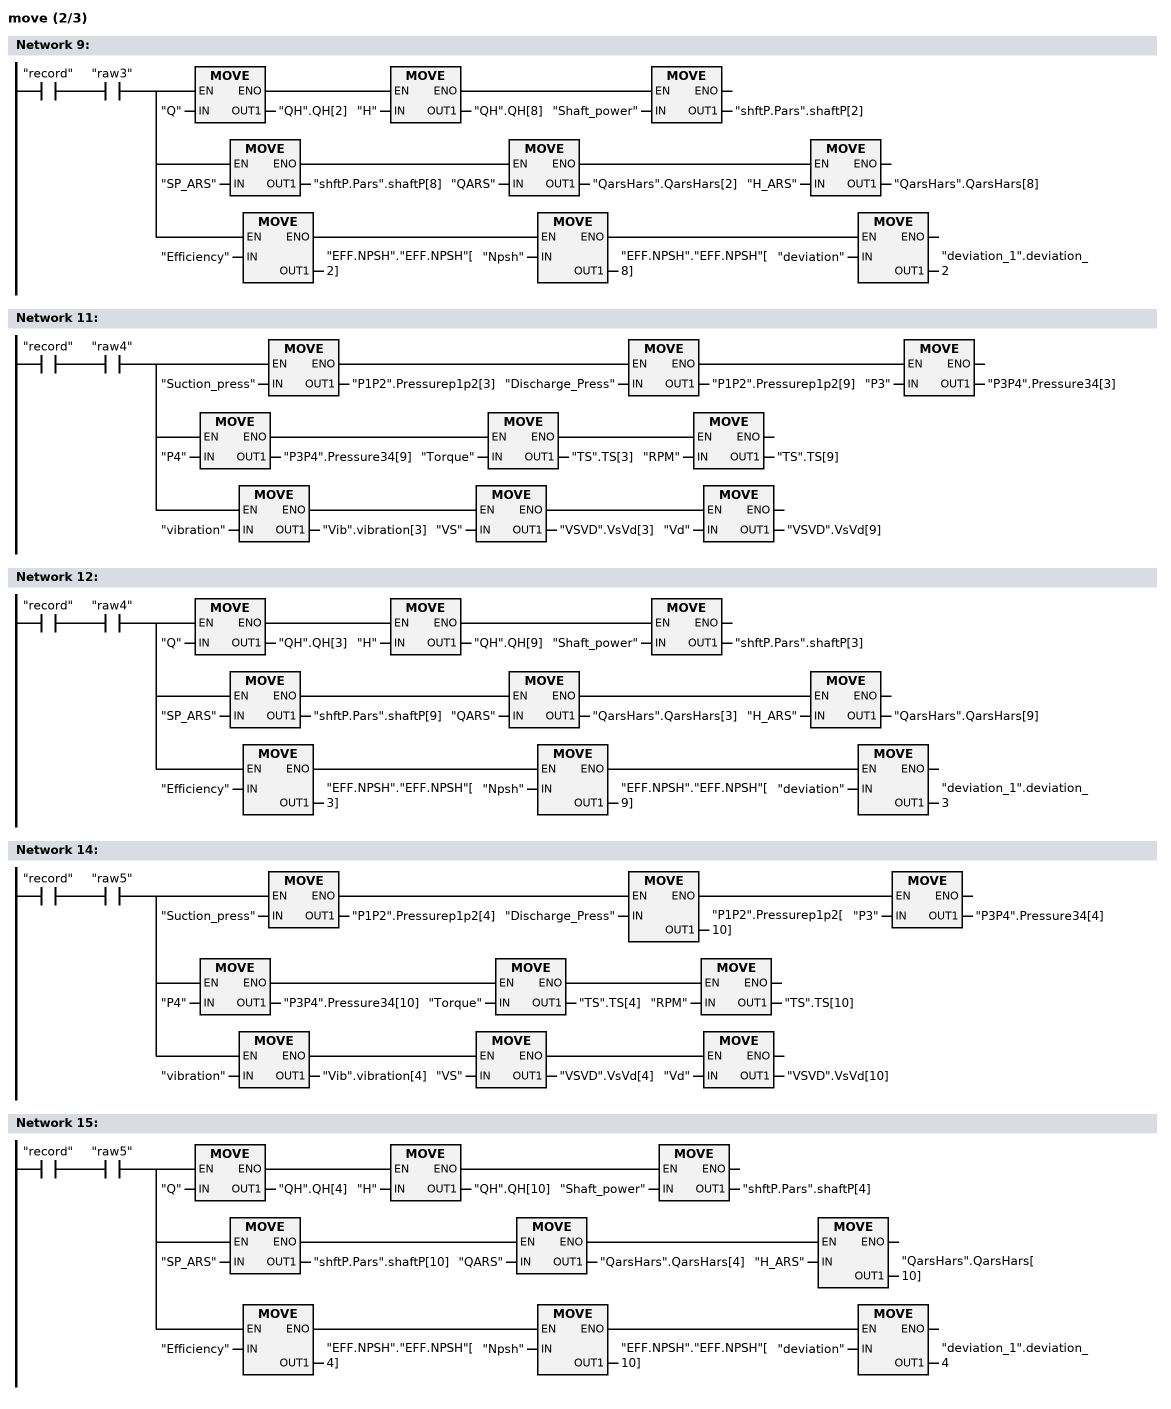
   RUNG wire#powerrail
      Contact( "record" )
      Contact( "raw3" )
      wire#w1
      Move(in := "Q", out1 => "QH".QH[2])
      Move(in := "H", out1 => "QH".QH[8])
      Move(in := "Shaft_power", out1 => "shftP.Pars".shaftP[2])
   END_RUNG
   RUNG wire#w1
      Move(in := "SP_ARS", out1 => "shftP.Pars".shaftP[8])
      Move(in := "QARS", out1 => "QarsHars".QarsHars[2])
      Move(in := "H_ARS", out1 => "QarsHars".QarsHars[8])
   END_RUNG
   RUNG wire#w1
      Move(in := "Efficiency", out1 => "EFF.NPSH"."EFF.NPSH"[2])
      Move(in := "Npsh", out1 => "EFF.NPSH"."EFF.NPSH"[8])
      Move(in := "deviation", out1 => "deviation_1".deviation_2)
   END_RUNG
   // the same network as SCL:
   IF "record" AND "raw3" THEN
       "QH".QH[2] := "Q";
       "QH".QH[8] := "H";
       "shftP.Pars".shaftP[2] := "Shaft_power";
       "shftP.Pars".shaftP[8] := "SP_ARS";
       "QarsHars".QarsHars[2] := "QARS";
       "QarsHars".QarsHars[8] := "H_ARS";
       "EFF.NPSH"."EFF.NPSH"[2] := "Efficiency";
       "EFF.NPSH"."EFF.NPSH"[8] := "Npsh";
       "deviation_1".deviation_2 := "deviation";
   END_IF;
END_REGION

REGION Network 11
   RUNG wire#powerrail
      Contact( "record" )
      Contact( "raw4" )
      wire#w1
      Move(in := "Suction_press", out1 => "P1P2".Pressurep1p2[3])
      Move(in := "Discharge_Press", out1 => "P1P2".Pressurep1p2[9])
      Move(in := "P3", out1 => "P3P4".Pressure34[3])
   END_RUNG
   RUNG wire#w1
      Move(in := "P4", out1 => "P3P4".Pressure34[9])
      Move(in := "Torque", out1 => "TS".TS[3])
      Move(in := "RPM", out1 => "TS".TS[9])
   END_RUNG
   RUNG wire#w1
      Move(in := "vibration", out1 => "Vib".vibration[3])
      Move(in := "VS", out1 => "VSVD".VsVd[3])
      Move(in := "Vd", out1 => "VSVD".VsVd[9])
   END_RUNG
   // the same network as SCL:
   IF "record" AND "raw4" THEN
       "P1P2".Pressurep1p2[3] := "Suction_press";
       "P1P2".Pressurep1p2[9] := "Discharge_Press";
       "P3P4".Pressure34[3] := "P3";
       "P3P4".Pressure34[9] := "P4";
       "TS".TS[3] := "Torque";
       "TS".TS[9] := "RPM";
       "Vib".vibration[3] := "vibration";
       "VSVD".VsVd[3] := "VS";
       "VSVD".VsVd[9] := "Vd";
   END_IF;
END_REGION

REGION Network 12
   RUNG wire#powerrail
      Contact( "record" )
      Contact( "raw4" )
      wire#w1
      Move(in := "Q", out1 => "QH".QH[3])
      Move(in := "H", out1 => "QH".QH[9])
      Move(in := "Shaft_power", out1 => "shftP.Pars".shaftP[3])
   END_RUNG
   RUNG wire#w1
      Move(in := "SP_ARS", out1 => "shftP.Pars".shaftP[9])
      Move(in := "QARS", out1 => "QarsHars".QarsHars[3])
      Move(in := "H_ARS", out1 => "QarsHars".QarsHars[9])
   END_RUNG
   RUNG wire#w1
      Move(in := "Efficiency", out1 => "EFF.NPSH"."EFF.NPSH"[3])
      Move(in := "Npsh", out1 => "EFF.NPSH"."EFF.NPSH"[9])
      Move(in := "deviation", out1 => "deviation_1".deviation_3)
   END_RUNG
   // the same network as SCL:
   IF "record" AND "raw4" THEN
       "QH".QH[3] := "Q";
       "QH".QH[9] := "H";
       "shftP.Pars".shaftP[3] := "Shaft_power";
       "shftP.Pars".shaftP[9] := "SP_ARS";
       "QarsHars".QarsHars[3] := "QARS";
       "QarsHars".QarsHars[9] := "H_ARS";
       "EFF.NPSH"."EFF.NPSH"[3] := "Efficiency";
       "EFF.NPSH"."EFF.NPSH"[9] := "Npsh";
       "deviation_1".deviation_3 := "deviation";
   END_IF;
END_REGION

REGION Network 14
   RUNG wire#powerrail
      Contact( "record" )
      Contact( "raw5" )
      wire#w1
      Move(in := "Suction_press", out1 => "P1P2".Pressurep1p2[4])
      Move(in := "Discharge_Press", out1 => "P1P2".Pressurep1p2[10])
      Move(in := "P3", out1 => "P3P4".Pressure34[4])
   END_RUNG
   RUNG wire#w1
      Move(in := "P4", out1 => "P3P4".Pressure34[10])
      Move(in := "Torque", out1 => "TS".TS[4])
      Move(in := "RPM", out1 => "TS".TS[10])
   END_RUNG
   RUNG wire#w1
      Move(in := "vibration", out1 => "Vib".vibration[4])
      Move(in := "VS", out1 => "VSVD".VsVd[4])
      Move(in := "Vd", out1 => "VSVD".VsVd[10])
   END_RUNG
   // the same network as SCL:
   IF "record" AND "raw5" THEN
       "P1P2".Pressurep1p2[4] := "Suction_press";
       "P1P2".Pressurep1p2[10] := "Discharge_Press";
       "P3P4".Pressure34[4] := "P3";
       "P3P4".Pressure34[10] := "P4";
       "TS".TS[4] := "Torque";
       "TS".TS[10] := "RPM";
       "Vib".vibration[4] := "vibration";
       "VSVD".VsVd[4] := "VS";
       "VSVD".VsVd[10] := "Vd";
   END_IF;
END_REGION

REGION Network 15
   RUNG wire#powerrail
      Contact( "record" )
      Contact( "raw5" )
      wire#w1
      Move(in := "Q", out1 => "QH".QH[4])
      Move(in := "H", out1 => "QH".QH[10])
      Move(in := "Shaft_power", out1 => "shftP.Pars".shaftP[4])
   END_RUNG
   RUNG wire#w1
      Move(in := "SP_ARS", out1 => "shftP.Pars".shaftP[10])
      Move(in := "QARS", out1 => "QarsHars".QarsHars[4])
      Move(in := "H_ARS", out1 => "QarsHars".QarsHars[10])
   END_RUNG
   RUNG wire#w1
      Move(in := "Efficiency", out1 => "EFF.NPSH"."EFF.NPSH"[4])
      Move(in := "Npsh", out1 => "EFF.NPSH"."EFF.NPSH"[10])
      Move(in := "deviation", out1 => "deviation_1".deviation_4)
   END_RUNG
   // the same network as SCL:
   IF "record" AND "raw5" THEN
       "QH".QH[4] := "Q";
       "QH".QH[10] := "H";
       "shftP.Pars".shaftP[4] := "Shaft_power";
       "shftP.Pars".shaftP[10] := "SP_ARS";
       "QarsHars".QarsHars[4] := "QARS";
       "QarsHars".QarsHars[10] := "H_ARS";
       "EFF.NPSH"."EFF.NPSH"[4] := "Efficiency";
       "EFF.NPSH"."EFF.NPSH"[10] := "Npsh";
       "deviation_1".deviation_4 := "deviation";
   END_IF;
END_REGION

REGION Network 17
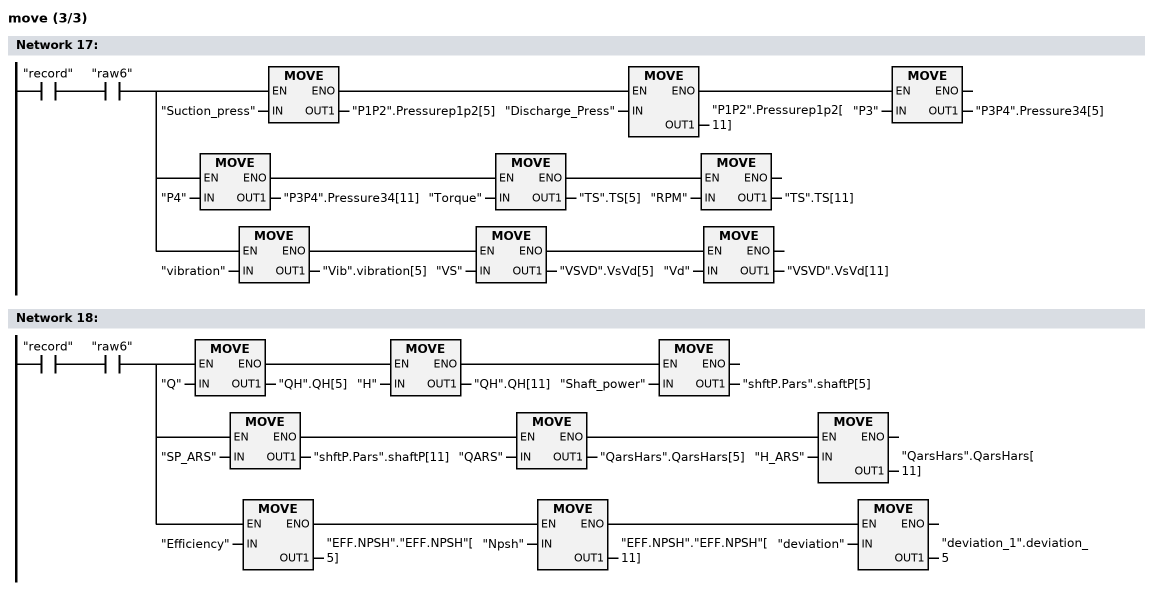
   RUNG wire#powerrail
      Contact( "record" )
      Contact( "raw6" )
      wire#w1
      Move(in := "Suction_press", out1 => "P1P2".Pressurep1p2[5])
      Move(in := "Discharge_Press", out1 => "P1P2".Pressurep1p2[11])
      Move(in := "P3", out1 => "P3P4".Pressure34[5])
   END_RUNG
   RUNG wire#w1
      Move(in := "P4", out1 => "P3P4".Pressure34[11])
      Move(in := "Torque", out1 => "TS".TS[5])
      Move(in := "RPM", out1 => "TS".TS[11])
   END_RUNG
   RUNG wire#w1
      Move(in := "vibration", out1 => "Vib".vibration[5])
      Move(in := "VS", out1 => "VSVD".VsVd[5])
      Move(in := "Vd", out1 => "VSVD".VsVd[11])
   END_RUNG
   // the same network as SCL:
   IF "record" AND "raw6" THEN
       "P1P2".Pressurep1p2[5] := "Suction_press";
       "P1P2".Pressurep1p2[11] := "Discharge_Press";
       "P3P4".Pressure34[5] := "P3";
       "P3P4".Pressure34[11] := "P4";
       "TS".TS[5] := "Torque";
       "TS".TS[11] := "RPM";
       "Vib".vibration[5] := "vibration";
       "VSVD".VsVd[5] := "VS";
       "VSVD".VsVd[11] := "Vd";
   END_IF;
END_REGION

REGION Network 18
   RUNG wire#powerrail
      Contact( "record" )
      Contact( "raw6" )
      wire#w1
      Move(in := "Q", out1 => "QH".QH[5])
      Move(in := "H", out1 => "QH".QH[11])
      Move(in := "Shaft_power", out1 => "shftP.Pars".shaftP[5])
   END_RUNG
   RUNG wire#w1
      Move(in := "SP_ARS", out1 => "shftP.Pars".shaftP[11])
      Move(in := "QARS", out1 => "QarsHars".QarsHars[5])
      Move(in := "H_ARS", out1 => "QarsHars".QarsHars[11])
   END_RUNG
   RUNG wire#w1
      Move(in := "Efficiency", out1 => "EFF.NPSH"."EFF.NPSH"[5])
      Move(in := "Npsh", out1 => "EFF.NPSH"."EFF.NPSH"[11])
      Move(in := "deviation", out1 => "deviation_1".deviation_5)
   END_RUNG
   // the same network as SCL:
   IF "record" AND "raw6" THEN
       "QH".QH[5] := "Q";
       "QH".QH[11] := "H";
       "shftP.Pars".shaftP[5] := "Shaft_power";
       "shftP.Pars".shaftP[11] := "SP_ARS";
       "QarsHars".QarsHars[5] := "QARS";
       "QarsHars".QarsHars[11] := "H_ARS";
       "EFF.NPSH"."EFF.NPSH"[5] := "Efficiency";
       "EFF.NPSH"."EFF.NPSH"[11] := "Npsh";
       "deviation_1".deviation_5 := "deviation";
   END_IF;
END_REGION
END_FUNCTION

FUNCTION "stepper" : Void   // FC5, LAD
{ S7_Optimized_Access := 'TRUE' }
VERSION : 0.1
BEGIN

REGION Network 1
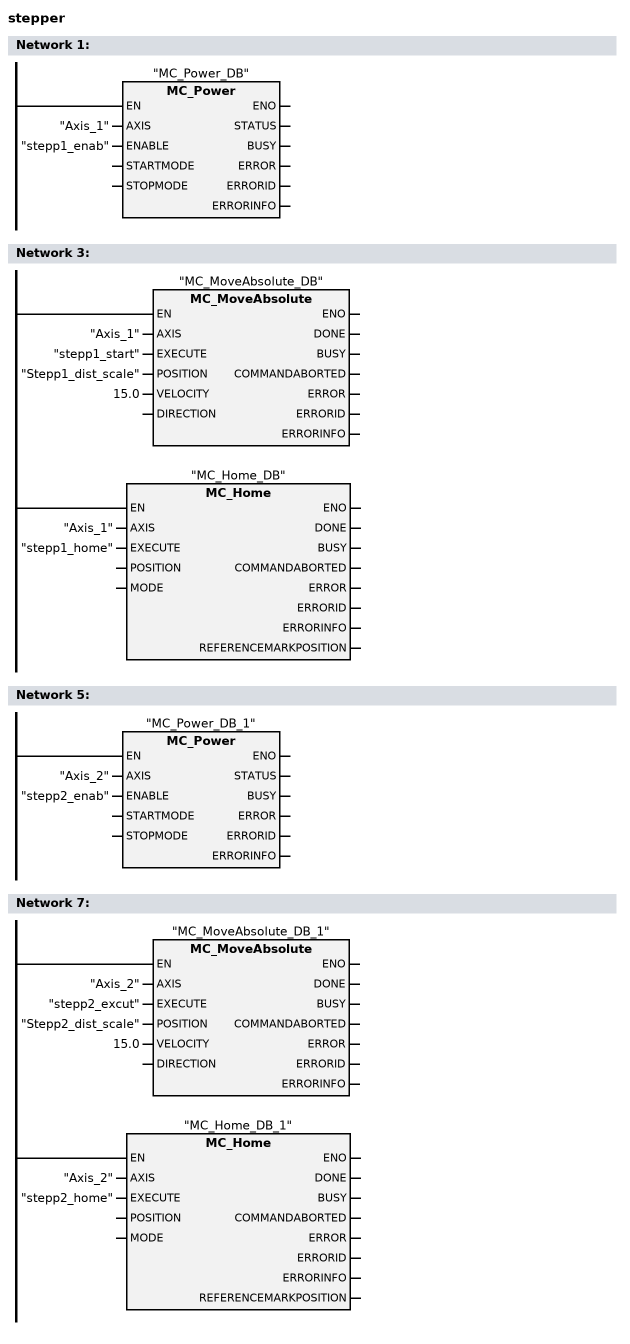
   "MC_Power_DB"(Axis := "Axis_1", Enable := "stepp1_enab");   // MC_Power
END_REGION

REGION Network 3
   "MC_MoveAbsolute_DB"(Axis := "Axis_1",   // MC_MoveAbsolute
                        Execute := "stepp1_start",
                        Position := "Stepp1_dist_scale",
                        Velocity := 15.0);
   "MC_Home_DB"(Axis := "Axis_1", Execute := "stepp1_home");   // MC_Home
END_REGION

REGION Network 5
   "MC_Power_DB_1"(Axis := "Axis_2", Enable := "stepp2_enab");   // MC_Power
END_REGION

REGION Network 7
   "MC_MoveAbsolute_DB_1"(Axis := "Axis_2",   // MC_MoveAbsolute
                          Execute := "stepp2_excut",
                          Position := "Stepp2_dist_scale",
                          Velocity := 15.0);
   "MC_Home_DB_1"(Axis := "Axis_2", Execute := "stepp2_home");   // MC_Home
END_REGION
END_FUNCTION

FUNCTION "clear" : Void   // FC6, LAD
{ S7_Optimized_Access := 'TRUE' }
VERSION : 0.1
BEGIN

REGION Network 2
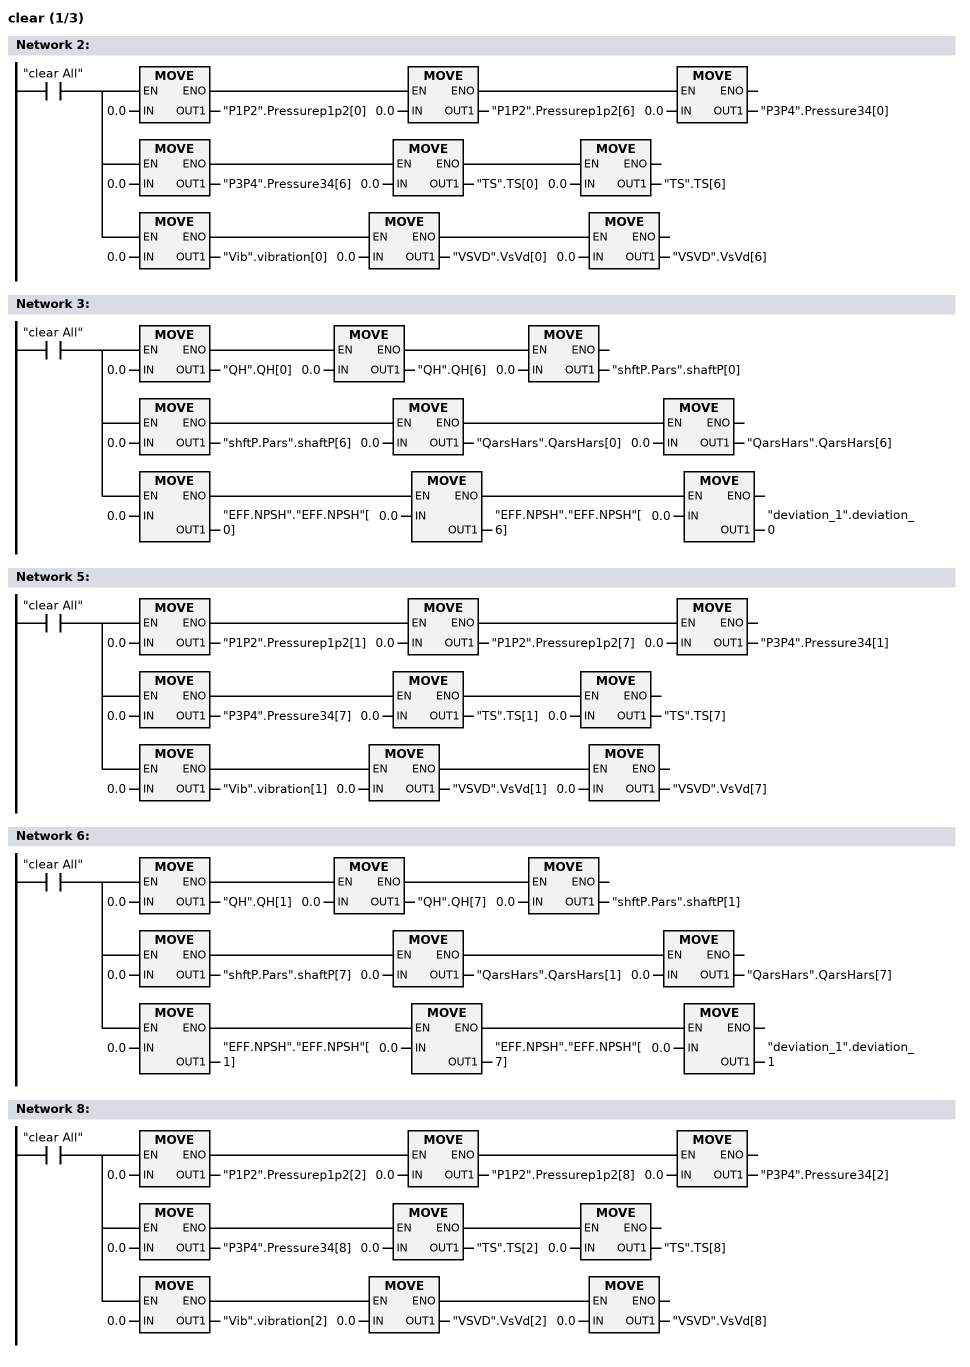
   RUNG wire#powerrail
      Contact( "clear All" )
      wire#w1
      Move(in := 0.0, out1 => "P1P2".Pressurep1p2[0])
      Move(in := 0.0, out1 => "P1P2".Pressurep1p2[6])
      Move(in := 0.0, out1 => "P3P4".Pressure34[0])
   END_RUNG
   RUNG wire#w1
      Move(in := 0.0, out1 => "P3P4".Pressure34[6])
      Move(in := 0.0, out1 => "TS".TS[0])
      Move(in := 0.0, out1 => "TS".TS[6])
   END_RUNG
   RUNG wire#w1
      Move(in := 0.0, out1 => "Vib".vibration[0])
      Move(in := 0.0, out1 => "VSVD".VsVd[0])
      Move(in := 0.0, out1 => "VSVD".VsVd[6])
   END_RUNG
   // the same network as SCL:
   IF "clear All" THEN
       "P1P2".Pressurep1p2[0] := 0.0;
       "P1P2".Pressurep1p2[6] := 0.0;
       "P3P4".Pressure34[0] := 0.0;
       "P3P4".Pressure34[6] := 0.0;
       "TS".TS[0] := 0.0;
       "TS".TS[6] := 0.0;
       "Vib".vibration[0] := 0.0;
       "VSVD".VsVd[0] := 0.0;
       "VSVD".VsVd[6] := 0.0;
   END_IF;
END_REGION

REGION Network 3
   RUNG wire#powerrail
      Contact( "clear All" )
      wire#w1
      Move(in := 0.0, out1 => "QH".QH[0])
      Move(in := 0.0, out1 => "QH".QH[6])
      Move(in := 0.0, out1 => "shftP.Pars".shaftP[0])
   END_RUNG
   RUNG wire#w1
      Move(in := 0.0, out1 => "shftP.Pars".shaftP[6])
      Move(in := 0.0, out1 => "QarsHars".QarsHars[0])
      Move(in := 0.0, out1 => "QarsHars".QarsHars[6])
   END_RUNG
   RUNG wire#w1
      Move(in := 0.0, out1 => "EFF.NPSH"."EFF.NPSH"[0])
      Move(in := 0.0, out1 => "EFF.NPSH"."EFF.NPSH"[6])
      Move(in := 0.0, out1 => "deviation_1".deviation_0)
   END_RUNG
   // the same network as SCL:
   IF "clear All" THEN
       "QH".QH[0] := 0.0;
       "QH".QH[6] := 0.0;
       "shftP.Pars".shaftP[0] := 0.0;
       "shftP.Pars".shaftP[6] := 0.0;
       "QarsHars".QarsHars[0] := 0.0;
       "QarsHars".QarsHars[6] := 0.0;
       "EFF.NPSH"."EFF.NPSH"[0] := 0.0;
       "EFF.NPSH"."EFF.NPSH"[6] := 0.0;
       "deviation_1".deviation_0 := 0.0;
   END_IF;
END_REGION

REGION Network 5
   RUNG wire#powerrail
      Contact( "clear All" )
      wire#w1
      Move(in := 0.0, out1 => "P1P2".Pressurep1p2[1])
      Move(in := 0.0, out1 => "P1P2".Pressurep1p2[7])
      Move(in := 0.0, out1 => "P3P4".Pressure34[1])
   END_RUNG
   RUNG wire#w1
      Move(in := 0.0, out1 => "P3P4".Pressure34[7])
      Move(in := 0.0, out1 => "TS".TS[1])
      Move(in := 0.0, out1 => "TS".TS[7])
   END_RUNG
   RUNG wire#w1
      Move(in := 0.0, out1 => "Vib".vibration[1])
      Move(in := 0.0, out1 => "VSVD".VsVd[1])
      Move(in := 0.0, out1 => "VSVD".VsVd[7])
   END_RUNG
   // the same network as SCL:
   IF "clear All" THEN
       "P1P2".Pressurep1p2[1] := 0.0;
       "P1P2".Pressurep1p2[7] := 0.0;
       "P3P4".Pressure34[1] := 0.0;
       "P3P4".Pressure34[7] := 0.0;
       "TS".TS[1] := 0.0;
       "TS".TS[7] := 0.0;
       "Vib".vibration[1] := 0.0;
       "VSVD".VsVd[1] := 0.0;
       "VSVD".VsVd[7] := 0.0;
   END_IF;
END_REGION

REGION Network 6
   RUNG wire#powerrail
      Contact( "clear All" )
      wire#w1
      Move(in := 0.0, out1 => "QH".QH[1])
      Move(in := 0.0, out1 => "QH".QH[7])
      Move(in := 0.0, out1 => "shftP.Pars".shaftP[1])
   END_RUNG
   RUNG wire#w1
      Move(in := 0.0, out1 => "shftP.Pars".shaftP[7])
      Move(in := 0.0, out1 => "QarsHars".QarsHars[1])
      Move(in := 0.0, out1 => "QarsHars".QarsHars[7])
   END_RUNG
   RUNG wire#w1
      Move(in := 0.0, out1 => "EFF.NPSH"."EFF.NPSH"[1])
      Move(in := 0.0, out1 => "EFF.NPSH"."EFF.NPSH"[7])
      Move(in := 0.0, out1 => "deviation_1".deviation_1)
   END_RUNG
   // the same network as SCL:
   IF "clear All" THEN
       "QH".QH[1] := 0.0;
       "QH".QH[7] := 0.0;
       "shftP.Pars".shaftP[1] := 0.0;
       "shftP.Pars".shaftP[7] := 0.0;
       "QarsHars".QarsHars[1] := 0.0;
       "QarsHars".QarsHars[7] := 0.0;
       "EFF.NPSH"."EFF.NPSH"[1] := 0.0;
       "EFF.NPSH"."EFF.NPSH"[7] := 0.0;
       "deviation_1".deviation_1 := 0.0;
   END_IF;
END_REGION

REGION Network 8
   RUNG wire#powerrail
      Contact( "clear All" )
      wire#w1
      Move(in := 0.0, out1 => "P1P2".Pressurep1p2[2])
      Move(in := 0.0, out1 => "P1P2".Pressurep1p2[8])
      Move(in := 0.0, out1 => "P3P4".Pressure34[2])
   END_RUNG
   RUNG wire#w1
      Move(in := 0.0, out1 => "P3P4".Pressure34[8])
      Move(in := 0.0, out1 => "TS".TS[2])
      Move(in := 0.0, out1 => "TS".TS[8])
   END_RUNG
   RUNG wire#w1
      Move(in := 0.0, out1 => "Vib".vibration[2])
      Move(in := 0.0, out1 => "VSVD".VsVd[2])
      Move(in := 0.0, out1 => "VSVD".VsVd[8])
   END_RUNG
   // the same network as SCL:
   IF "clear All" THEN
       "P1P2".Pressurep1p2[2] := 0.0;
       "P1P2".Pressurep1p2[8] := 0.0;
       "P3P4".Pressure34[2] := 0.0;
       "P3P4".Pressure34[8] := 0.0;
       "TS".TS[2] := 0.0;
       "TS".TS[8] := 0.0;
       "Vib".vibration[2] := 0.0;
       "VSVD".VsVd[2] := 0.0;
       "VSVD".VsVd[8] := 0.0;
   END_IF;
END_REGION

REGION Network 9
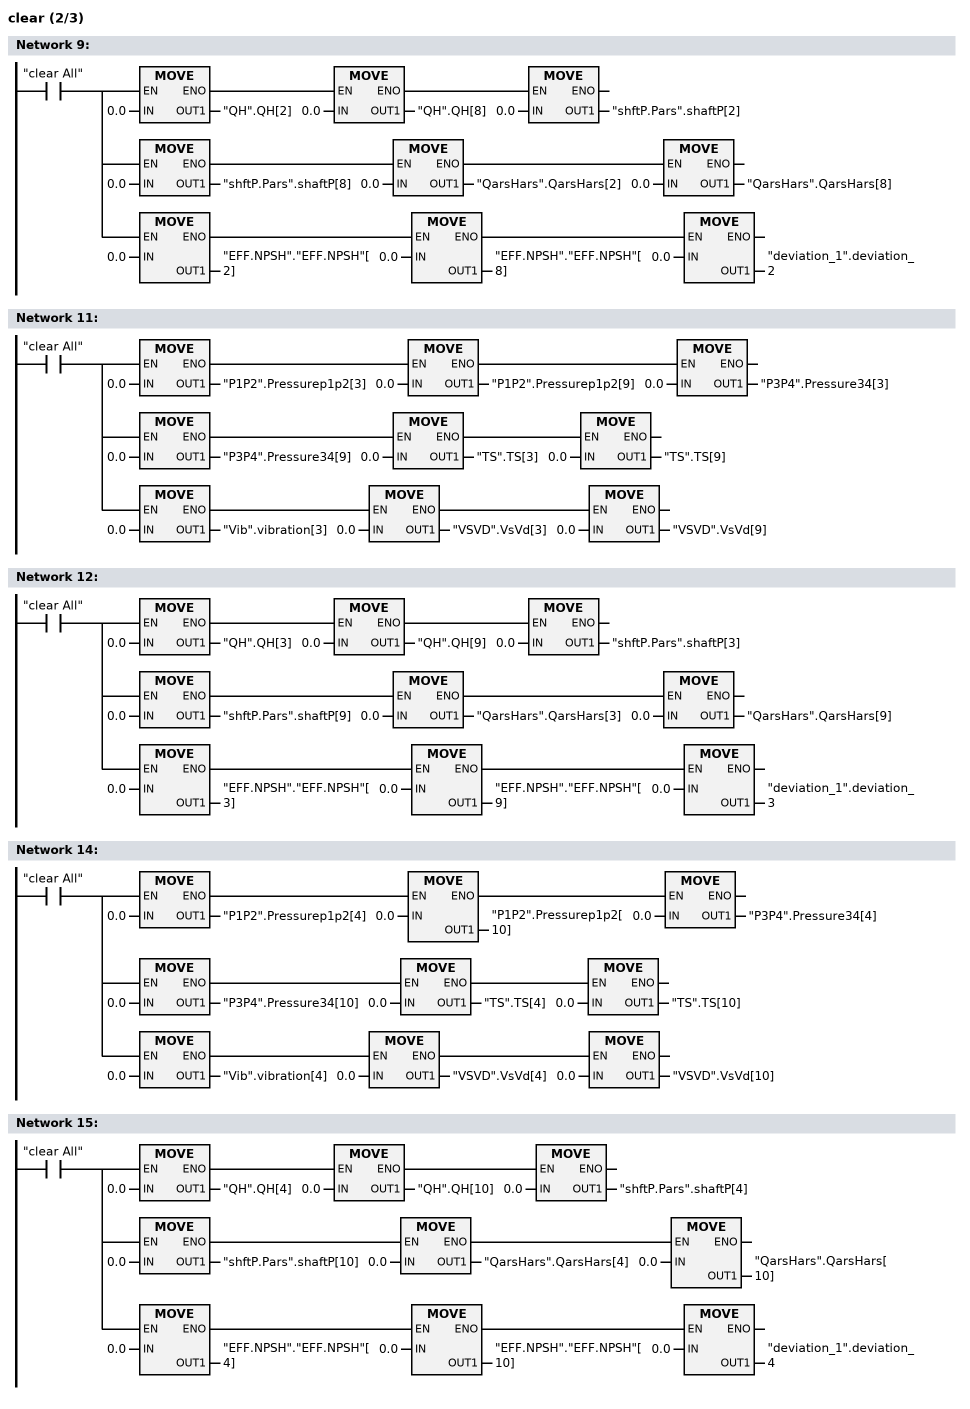
   RUNG wire#powerrail
      Contact( "clear All" )
      wire#w1
      Move(in := 0.0, out1 => "QH".QH[2])
      Move(in := 0.0, out1 => "QH".QH[8])
      Move(in := 0.0, out1 => "shftP.Pars".shaftP[2])
   END_RUNG
   RUNG wire#w1
      Move(in := 0.0, out1 => "shftP.Pars".shaftP[8])
      Move(in := 0.0, out1 => "QarsHars".QarsHars[2])
      Move(in := 0.0, out1 => "QarsHars".QarsHars[8])
   END_RUNG
   RUNG wire#w1
      Move(in := 0.0, out1 => "EFF.NPSH"."EFF.NPSH"[2])
      Move(in := 0.0, out1 => "EFF.NPSH"."EFF.NPSH"[8])
      Move(in := 0.0, out1 => "deviation_1".deviation_2)
   END_RUNG
   // the same network as SCL:
   IF "clear All" THEN
       "QH".QH[2] := 0.0;
       "QH".QH[8] := 0.0;
       "shftP.Pars".shaftP[2] := 0.0;
       "shftP.Pars".shaftP[8] := 0.0;
       "QarsHars".QarsHars[2] := 0.0;
       "QarsHars".QarsHars[8] := 0.0;
       "EFF.NPSH"."EFF.NPSH"[2] := 0.0;
       "EFF.NPSH"."EFF.NPSH"[8] := 0.0;
       "deviation_1".deviation_2 := 0.0;
   END_IF;
END_REGION

REGION Network 11
   RUNG wire#powerrail
      Contact( "clear All" )
      wire#w1
      Move(in := 0.0, out1 => "P1P2".Pressurep1p2[3])
      Move(in := 0.0, out1 => "P1P2".Pressurep1p2[9])
      Move(in := 0.0, out1 => "P3P4".Pressure34[3])
   END_RUNG
   RUNG wire#w1
      Move(in := 0.0, out1 => "P3P4".Pressure34[9])
      Move(in := 0.0, out1 => "TS".TS[3])
      Move(in := 0.0, out1 => "TS".TS[9])
   END_RUNG
   RUNG wire#w1
      Move(in := 0.0, out1 => "Vib".vibration[3])
      Move(in := 0.0, out1 => "VSVD".VsVd[3])
      Move(in := 0.0, out1 => "VSVD".VsVd[9])
   END_RUNG
   // the same network as SCL:
   IF "clear All" THEN
       "P1P2".Pressurep1p2[3] := 0.0;
       "P1P2".Pressurep1p2[9] := 0.0;
       "P3P4".Pressure34[3] := 0.0;
       "P3P4".Pressure34[9] := 0.0;
       "TS".TS[3] := 0.0;
       "TS".TS[9] := 0.0;
       "Vib".vibration[3] := 0.0;
       "VSVD".VsVd[3] := 0.0;
       "VSVD".VsVd[9] := 0.0;
   END_IF;
END_REGION

REGION Network 12
   RUNG wire#powerrail
      Contact( "clear All" )
      wire#w1
      Move(in := 0.0, out1 => "QH".QH[3])
      Move(in := 0.0, out1 => "QH".QH[9])
      Move(in := 0.0, out1 => "shftP.Pars".shaftP[3])
   END_RUNG
   RUNG wire#w1
      Move(in := 0.0, out1 => "shftP.Pars".shaftP[9])
      Move(in := 0.0, out1 => "QarsHars".QarsHars[3])
      Move(in := 0.0, out1 => "QarsHars".QarsHars[9])
   END_RUNG
   RUNG wire#w1
      Move(in := 0.0, out1 => "EFF.NPSH"."EFF.NPSH"[3])
      Move(in := 0.0, out1 => "EFF.NPSH"."EFF.NPSH"[9])
      Move(in := 0.0, out1 => "deviation_1".deviation_3)
   END_RUNG
   // the same network as SCL:
   IF "clear All" THEN
       "QH".QH[3] := 0.0;
       "QH".QH[9] := 0.0;
       "shftP.Pars".shaftP[3] := 0.0;
       "shftP.Pars".shaftP[9] := 0.0;
       "QarsHars".QarsHars[3] := 0.0;
       "QarsHars".QarsHars[9] := 0.0;
       "EFF.NPSH"."EFF.NPSH"[3] := 0.0;
       "EFF.NPSH"."EFF.NPSH"[9] := 0.0;
       "deviation_1".deviation_3 := 0.0;
   END_IF;
END_REGION

REGION Network 14
   RUNG wire#powerrail
      Contact( "clear All" )
      wire#w1
      Move(in := 0.0, out1 => "P1P2".Pressurep1p2[4])
      Move(in := 0.0, out1 => "P1P2".Pressurep1p2[10])
      Move(in := 0.0, out1 => "P3P4".Pressure34[4])
   END_RUNG
   RUNG wire#w1
      Move(in := 0.0, out1 => "P3P4".Pressure34[10])
      Move(in := 0.0, out1 => "TS".TS[4])
      Move(in := 0.0, out1 => "TS".TS[10])
   END_RUNG
   RUNG wire#w1
      Move(in := 0.0, out1 => "Vib".vibration[4])
      Move(in := 0.0, out1 => "VSVD".VsVd[4])
      Move(in := 0.0, out1 => "VSVD".VsVd[10])
   END_RUNG
   // the same network as SCL:
   IF "clear All" THEN
       "P1P2".Pressurep1p2[4] := 0.0;
       "P1P2".Pressurep1p2[10] := 0.0;
       "P3P4".Pressure34[4] := 0.0;
       "P3P4".Pressure34[10] := 0.0;
       "TS".TS[4] := 0.0;
       "TS".TS[10] := 0.0;
       "Vib".vibration[4] := 0.0;
       "VSVD".VsVd[4] := 0.0;
       "VSVD".VsVd[10] := 0.0;
   END_IF;
END_REGION

REGION Network 15
   RUNG wire#powerrail
      Contact( "clear All" )
      wire#w1
      Move(in := 0.0, out1 => "QH".QH[4])
      Move(in := 0.0, out1 => "QH".QH[10])
      Move(in := 0.0, out1 => "shftP.Pars".shaftP[4])
   END_RUNG
   RUNG wire#w1
      Move(in := 0.0, out1 => "shftP.Pars".shaftP[10])
      Move(in := 0.0, out1 => "QarsHars".QarsHars[4])
      Move(in := 0.0, out1 => "QarsHars".QarsHars[10])
   END_RUNG
   RUNG wire#w1
      Move(in := 0.0, out1 => "EFF.NPSH"."EFF.NPSH"[4])
      Move(in := 0.0, out1 => "EFF.NPSH"."EFF.NPSH"[10])
      Move(in := 0.0, out1 => "deviation_1".deviation_4)
   END_RUNG
   // the same network as SCL:
   IF "clear All" THEN
       "QH".QH[4] := 0.0;
       "QH".QH[10] := 0.0;
       "shftP.Pars".shaftP[4] := 0.0;
       "shftP.Pars".shaftP[10] := 0.0;
       "QarsHars".QarsHars[4] := 0.0;
       "QarsHars".QarsHars[10] := 0.0;
       "EFF.NPSH"."EFF.NPSH"[4] := 0.0;
       "EFF.NPSH"."EFF.NPSH"[10] := 0.0;
       "deviation_1".deviation_4 := 0.0;
   END_IF;
END_REGION

REGION Network 17
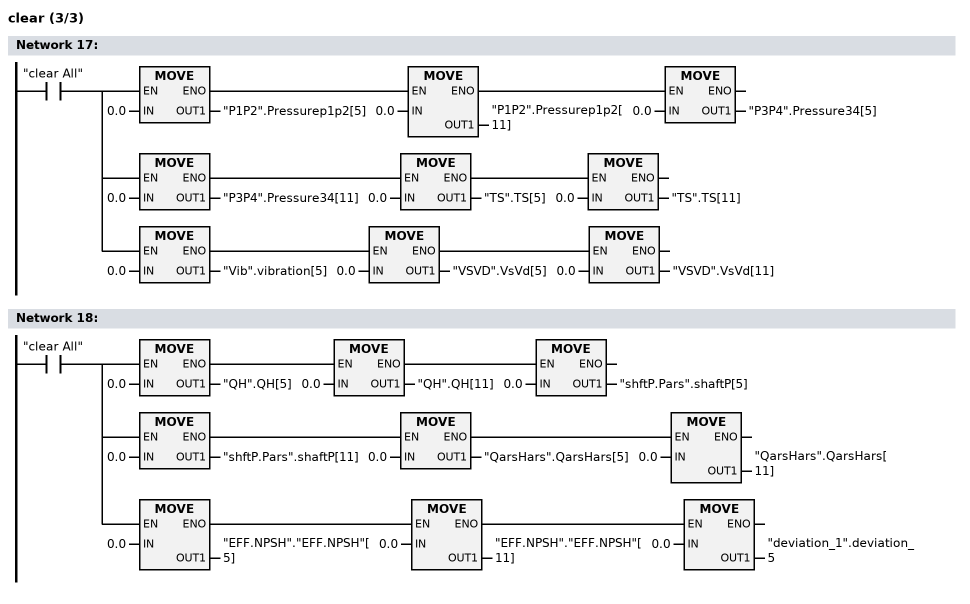
   RUNG wire#powerrail
      Contact( "clear All" )
      wire#w1
      Move(in := 0.0, out1 => "P1P2".Pressurep1p2[5])
      Move(in := 0.0, out1 => "P1P2".Pressurep1p2[11])
      Move(in := 0.0, out1 => "P3P4".Pressure34[5])
   END_RUNG
   RUNG wire#w1
      Move(in := 0.0, out1 => "P3P4".Pressure34[11])
      Move(in := 0.0, out1 => "TS".TS[5])
      Move(in := 0.0, out1 => "TS".TS[11])
   END_RUNG
   RUNG wire#w1
      Move(in := 0.0, out1 => "Vib".vibration[5])
      Move(in := 0.0, out1 => "VSVD".VsVd[5])
      Move(in := 0.0, out1 => "VSVD".VsVd[11])
   END_RUNG
   // the same network as SCL:
   IF "clear All" THEN
       "P1P2".Pressurep1p2[5] := 0.0;
       "P1P2".Pressurep1p2[11] := 0.0;
       "P3P4".Pressure34[5] := 0.0;
       "P3P4".Pressure34[11] := 0.0;
       "TS".TS[5] := 0.0;
       "TS".TS[11] := 0.0;
       "Vib".vibration[5] := 0.0;
       "VSVD".VsVd[5] := 0.0;
       "VSVD".VsVd[11] := 0.0;
   END_IF;
END_REGION

REGION Network 18
   RUNG wire#powerrail
      Contact( "clear All" )
      wire#w1
      Move(in := 0.0, out1 => "QH".QH[5])
      Move(in := 0.0, out1 => "QH".QH[11])
      Move(in := 0.0, out1 => "shftP.Pars".shaftP[5])
   END_RUNG
   RUNG wire#w1
      Move(in := 0.0, out1 => "shftP.Pars".shaftP[11])
      Move(in := 0.0, out1 => "QarsHars".QarsHars[5])
      Move(in := 0.0, out1 => "QarsHars".QarsHars[11])
   END_RUNG
   RUNG wire#w1
      Move(in := 0.0, out1 => "EFF.NPSH"."EFF.NPSH"[5])
      Move(in := 0.0, out1 => "EFF.NPSH"."EFF.NPSH"[11])
      Move(in := 0.0, out1 => "deviation_1".deviation_5)
   END_RUNG
   // the same network as SCL:
   IF "clear All" THEN
       "QH".QH[5] := 0.0;
       "QH".QH[11] := 0.0;
       "shftP.Pars".shaftP[5] := 0.0;
       "shftP.Pars".shaftP[11] := 0.0;
       "QarsHars".QarsHars[5] := 0.0;
       "QarsHars".QarsHars[11] := 0.0;
       "EFF.NPSH"."EFF.NPSH"[5] := 0.0;
       "EFF.NPSH"."EFF.NPSH"[11] := 0.0;
       "deviation_1".deviation_5 := 0.0;
   END_IF;
END_REGION
END_FUNCTION

FUNCTION "move_2" : Void   // FC7, LAD
{ S7_Optimized_Access := 'TRUE' }
VERSION : 0.1
BEGIN

REGION Network 2
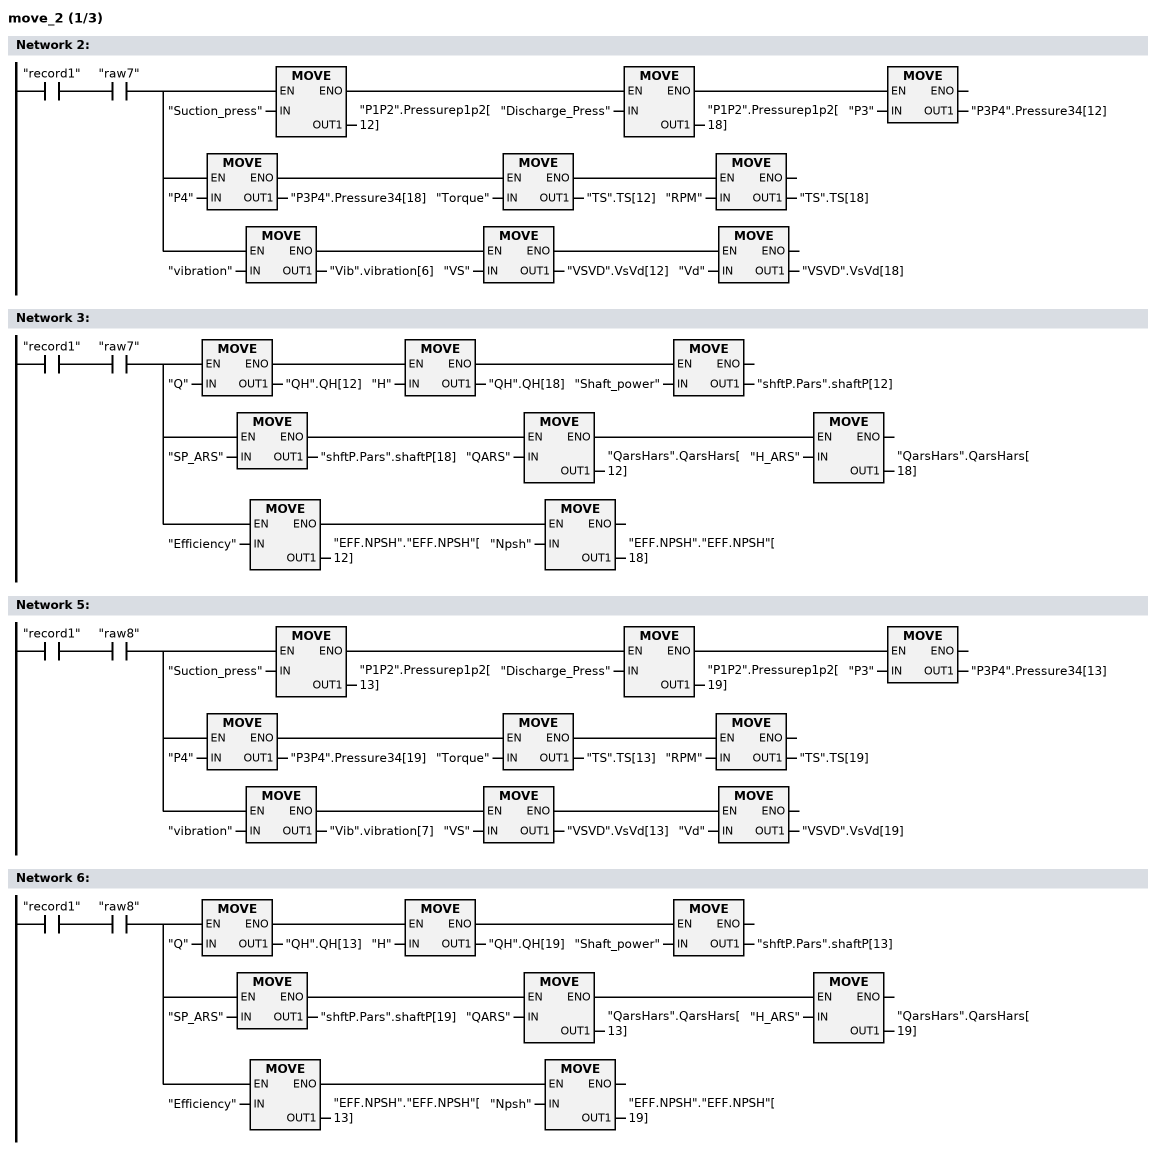
   RUNG wire#powerrail
      Contact( "record1" )
      Contact( "raw7" )
      wire#w1
      Move(in := "Suction_press", out1 => "P1P2".Pressurep1p2[12])
      Move(in := "Discharge_Press", out1 => "P1P2".Pressurep1p2[18])
      Move(in := "P3", out1 => "P3P4".Pressure34[12])
   END_RUNG
   RUNG wire#w1
      Move(in := "P4", out1 => "P3P4".Pressure34[18])
      Move(in := "Torque", out1 => "TS".TS[12])
      Move(in := "RPM", out1 => "TS".TS[18])
   END_RUNG
   RUNG wire#w1
      Move(in := "vibration", out1 => "Vib".vibration[6])
      Move(in := "VS", out1 => "VSVD".VsVd[12])
      Move(in := "Vd", out1 => "VSVD".VsVd[18])
   END_RUNG
   // the same network as SCL:
   IF "record1" AND "raw7" THEN
       "P1P2".Pressurep1p2[12] := "Suction_press";
       "P1P2".Pressurep1p2[18] := "Discharge_Press";
       "P3P4".Pressure34[12] := "P3";
       "P3P4".Pressure34[18] := "P4";
       "TS".TS[12] := "Torque";
       "TS".TS[18] := "RPM";
       "Vib".vibration[6] := "vibration";
       "VSVD".VsVd[12] := "VS";
       "VSVD".VsVd[18] := "Vd";
   END_IF;
END_REGION

REGION Network 3
   RUNG wire#powerrail
      Contact( "record1" )
      Contact( "raw7" )
      wire#w1
      Move(in := "Q", out1 => "QH".QH[12])
      Move(in := "H", out1 => "QH".QH[18])
      Move(in := "Shaft_power", out1 => "shftP.Pars".shaftP[12])
   END_RUNG
   RUNG wire#w1
      Move(in := "SP_ARS", out1 => "shftP.Pars".shaftP[18])
      Move(in := "QARS", out1 => "QarsHars".QarsHars[12])
      Move(in := "H_ARS", out1 => "QarsHars".QarsHars[18])
   END_RUNG
   RUNG wire#w1
      Move(in := "Efficiency", out1 => "EFF.NPSH"."EFF.NPSH"[12])
      Move(in := "Npsh", out1 => "EFF.NPSH"."EFF.NPSH"[18])
   END_RUNG
   // the same network as SCL:
   IF "record1" AND "raw7" THEN
       "QH".QH[12] := "Q";
       "QH".QH[18] := "H";
       "shftP.Pars".shaftP[12] := "Shaft_power";
       "shftP.Pars".shaftP[18] := "SP_ARS";
       "QarsHars".QarsHars[12] := "QARS";
       "QarsHars".QarsHars[18] := "H_ARS";
       "EFF.NPSH"."EFF.NPSH"[12] := "Efficiency";
       "EFF.NPSH"."EFF.NPSH"[18] := "Npsh";
   END_IF;
END_REGION

REGION Network 5
   RUNG wire#powerrail
      Contact( "record1" )
      Contact( "raw8" )
      wire#w1
      Move(in := "Suction_press", out1 => "P1P2".Pressurep1p2[13])
      Move(in := "Discharge_Press", out1 => "P1P2".Pressurep1p2[19])
      Move(in := "P3", out1 => "P3P4".Pressure34[13])
   END_RUNG
   RUNG wire#w1
      Move(in := "P4", out1 => "P3P4".Pressure34[19])
      Move(in := "Torque", out1 => "TS".TS[13])
      Move(in := "RPM", out1 => "TS".TS[19])
   END_RUNG
   RUNG wire#w1
      Move(in := "vibration", out1 => "Vib".vibration[7])
      Move(in := "VS", out1 => "VSVD".VsVd[13])
      Move(in := "Vd", out1 => "VSVD".VsVd[19])
   END_RUNG
   // the same network as SCL:
   IF "record1" AND "raw8" THEN
       "P1P2".Pressurep1p2[13] := "Suction_press";
       "P1P2".Pressurep1p2[19] := "Discharge_Press";
       "P3P4".Pressure34[13] := "P3";
       "P3P4".Pressure34[19] := "P4";
       "TS".TS[13] := "Torque";
       "TS".TS[19] := "RPM";
       "Vib".vibration[7] := "vibration";
       "VSVD".VsVd[13] := "VS";
       "VSVD".VsVd[19] := "Vd";
   END_IF;
END_REGION

REGION Network 6
   RUNG wire#powerrail
      Contact( "record1" )
      Contact( "raw8" )
      wire#w1
      Move(in := "Q", out1 => "QH".QH[13])
      Move(in := "H", out1 => "QH".QH[19])
      Move(in := "Shaft_power", out1 => "shftP.Pars".shaftP[13])
   END_RUNG
   RUNG wire#w1
      Move(in := "SP_ARS", out1 => "shftP.Pars".shaftP[19])
      Move(in := "QARS", out1 => "QarsHars".QarsHars[13])
      Move(in := "H_ARS", out1 => "QarsHars".QarsHars[19])
   END_RUNG
   RUNG wire#w1
      Move(in := "Efficiency", out1 => "EFF.NPSH"."EFF.NPSH"[13])
      Move(in := "Npsh", out1 => "EFF.NPSH"."EFF.NPSH"[19])
   END_RUNG
   // the same network as SCL:
   IF "record1" AND "raw8" THEN
       "QH".QH[13] := "Q";
       "QH".QH[19] := "H";
       "shftP.Pars".shaftP[13] := "Shaft_power";
       "shftP.Pars".shaftP[19] := "SP_ARS";
       "QarsHars".QarsHars[13] := "QARS";
       "QarsHars".QarsHars[19] := "H_ARS";
       "EFF.NPSH"."EFF.NPSH"[13] := "Efficiency";
       "EFF.NPSH"."EFF.NPSH"[19] := "Npsh";
   END_IF;
END_REGION

REGION Network 8
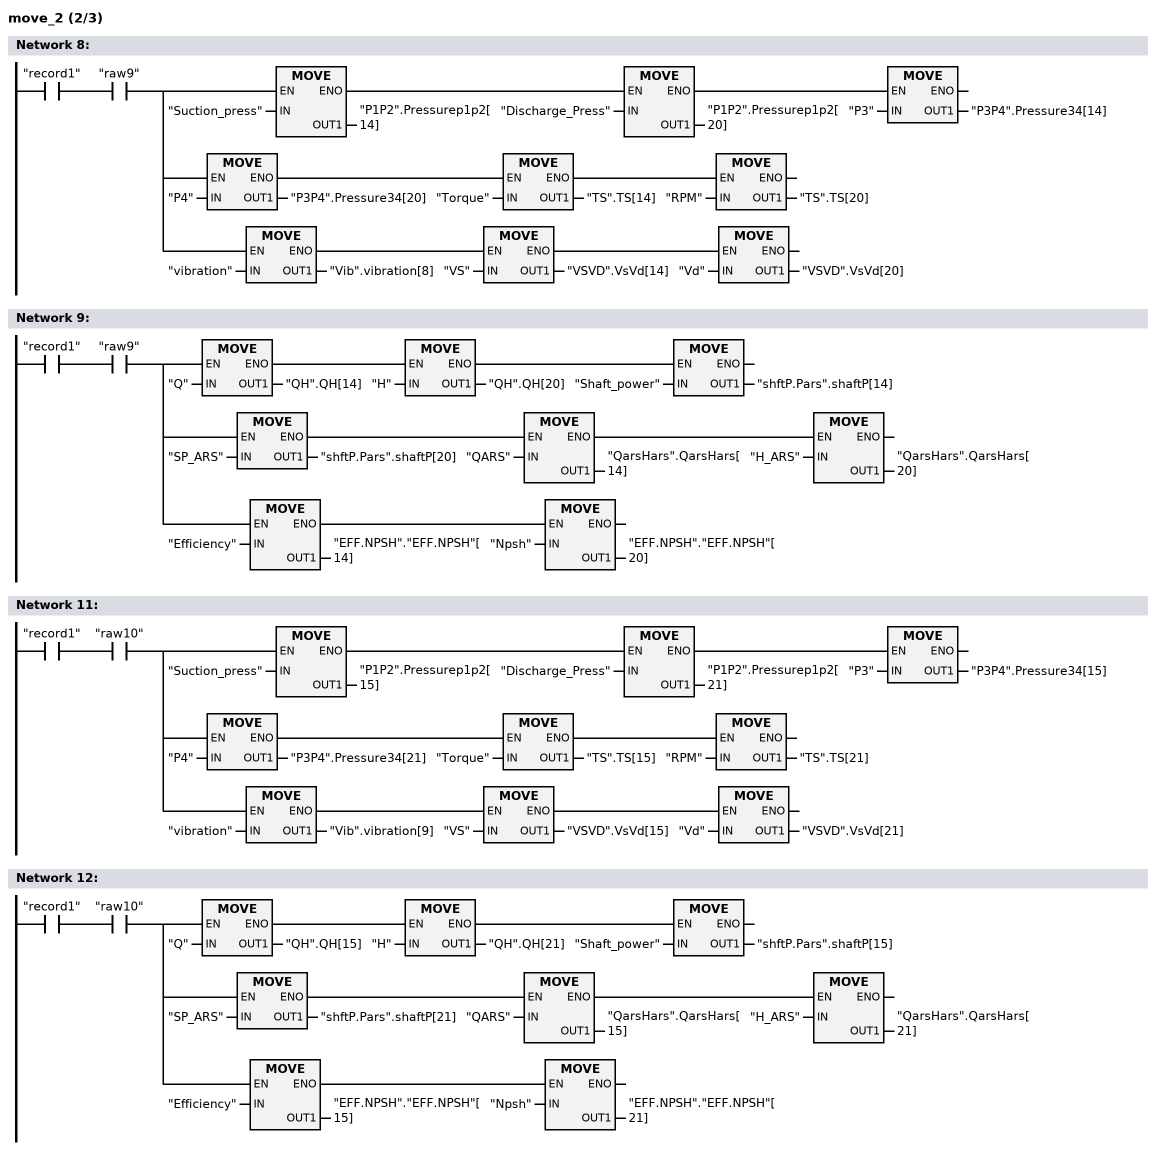
   RUNG wire#powerrail
      Contact( "record1" )
      Contact( "raw9" )
      wire#w1
      Move(in := "Suction_press", out1 => "P1P2".Pressurep1p2[14])
      Move(in := "Discharge_Press", out1 => "P1P2".Pressurep1p2[20])
      Move(in := "P3", out1 => "P3P4".Pressure34[14])
   END_RUNG
   RUNG wire#w1
      Move(in := "P4", out1 => "P3P4".Pressure34[20])
      Move(in := "Torque", out1 => "TS".TS[14])
      Move(in := "RPM", out1 => "TS".TS[20])
   END_RUNG
   RUNG wire#w1
      Move(in := "vibration", out1 => "Vib".vibration[8])
      Move(in := "VS", out1 => "VSVD".VsVd[14])
      Move(in := "Vd", out1 => "VSVD".VsVd[20])
   END_RUNG
   // the same network as SCL:
   IF "record1" AND "raw9" THEN
       "P1P2".Pressurep1p2[14] := "Suction_press";
       "P1P2".Pressurep1p2[20] := "Discharge_Press";
       "P3P4".Pressure34[14] := "P3";
       "P3P4".Pressure34[20] := "P4";
       "TS".TS[14] := "Torque";
       "TS".TS[20] := "RPM";
       "Vib".vibration[8] := "vibration";
       "VSVD".VsVd[14] := "VS";
       "VSVD".VsVd[20] := "Vd";
   END_IF;
END_REGION

REGION Network 9
   RUNG wire#powerrail
      Contact( "record1" )
      Contact( "raw9" )
      wire#w1
      Move(in := "Q", out1 => "QH".QH[14])
      Move(in := "H", out1 => "QH".QH[20])
      Move(in := "Shaft_power", out1 => "shftP.Pars".shaftP[14])
   END_RUNG
   RUNG wire#w1
      Move(in := "SP_ARS", out1 => "shftP.Pars".shaftP[20])
      Move(in := "QARS", out1 => "QarsHars".QarsHars[14])
      Move(in := "H_ARS", out1 => "QarsHars".QarsHars[20])
   END_RUNG
   RUNG wire#w1
      Move(in := "Efficiency", out1 => "EFF.NPSH"."EFF.NPSH"[14])
      Move(in := "Npsh", out1 => "EFF.NPSH"."EFF.NPSH"[20])
   END_RUNG
   // the same network as SCL:
   IF "record1" AND "raw9" THEN
       "QH".QH[14] := "Q";
       "QH".QH[20] := "H";
       "shftP.Pars".shaftP[14] := "Shaft_power";
       "shftP.Pars".shaftP[20] := "SP_ARS";
       "QarsHars".QarsHars[14] := "QARS";
       "QarsHars".QarsHars[20] := "H_ARS";
       "EFF.NPSH"."EFF.NPSH"[14] := "Efficiency";
       "EFF.NPSH"."EFF.NPSH"[20] := "Npsh";
   END_IF;
END_REGION

REGION Network 11
   RUNG wire#powerrail
      Contact( "record1" )
      Contact( "raw10" )
      wire#w1
      Move(in := "Suction_press", out1 => "P1P2".Pressurep1p2[15])
      Move(in := "Discharge_Press", out1 => "P1P2".Pressurep1p2[21])
      Move(in := "P3", out1 => "P3P4".Pressure34[15])
   END_RUNG
   RUNG wire#w1
      Move(in := "P4", out1 => "P3P4".Pressure34[21])
      Move(in := "Torque", out1 => "TS".TS[15])
      Move(in := "RPM", out1 => "TS".TS[21])
   END_RUNG
   RUNG wire#w1
      Move(in := "vibration", out1 => "Vib".vibration[9])
      Move(in := "VS", out1 => "VSVD".VsVd[15])
      Move(in := "Vd", out1 => "VSVD".VsVd[21])
   END_RUNG
   // the same network as SCL:
   IF "record1" AND "raw10" THEN
       "P1P2".Pressurep1p2[15] := "Suction_press";
       "P1P2".Pressurep1p2[21] := "Discharge_Press";
       "P3P4".Pressure34[15] := "P3";
       "P3P4".Pressure34[21] := "P4";
       "TS".TS[15] := "Torque";
       "TS".TS[21] := "RPM";
       "Vib".vibration[9] := "vibration";
       "VSVD".VsVd[15] := "VS";
       "VSVD".VsVd[21] := "Vd";
   END_IF;
END_REGION

REGION Network 12
   RUNG wire#powerrail
      Contact( "record1" )
      Contact( "raw10" )
      wire#w1
      Move(in := "Q", out1 => "QH".QH[15])
      Move(in := "H", out1 => "QH".QH[21])
      Move(in := "Shaft_power", out1 => "shftP.Pars".shaftP[15])
   END_RUNG
   RUNG wire#w1
      Move(in := "SP_ARS", out1 => "shftP.Pars".shaftP[21])
      Move(in := "QARS", out1 => "QarsHars".QarsHars[15])
      Move(in := "H_ARS", out1 => "QarsHars".QarsHars[21])
   END_RUNG
   RUNG wire#w1
      Move(in := "Efficiency", out1 => "EFF.NPSH"."EFF.NPSH"[15])
      Move(in := "Npsh", out1 => "EFF.NPSH"."EFF.NPSH"[21])
   END_RUNG
   // the same network as SCL:
   IF "record1" AND "raw10" THEN
       "QH".QH[15] := "Q";
       "QH".QH[21] := "H";
       "shftP.Pars".shaftP[15] := "Shaft_power";
       "shftP.Pars".shaftP[21] := "SP_ARS";
       "QarsHars".QarsHars[15] := "QARS";
       "QarsHars".QarsHars[21] := "H_ARS";
       "EFF.NPSH"."EFF.NPSH"[15] := "Efficiency";
       "EFF.NPSH"."EFF.NPSH"[21] := "Npsh";
   END_IF;
END_REGION

REGION Network 14
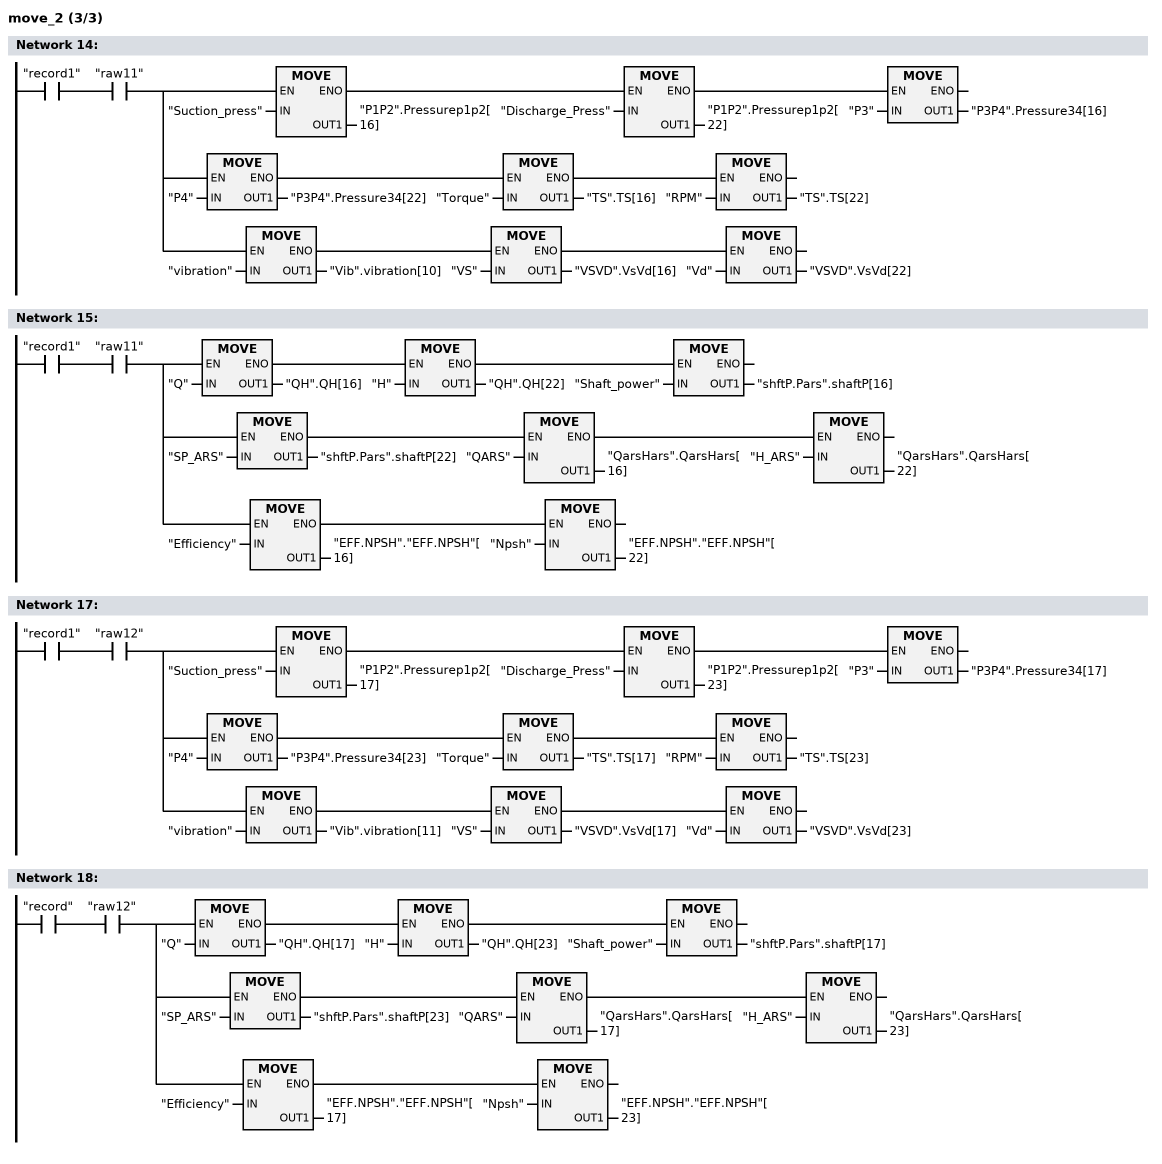
   RUNG wire#powerrail
      Contact( "record1" )
      Contact( "raw11" )
      wire#w1
      Move(in := "Suction_press", out1 => "P1P2".Pressurep1p2[16])
      Move(in := "Discharge_Press", out1 => "P1P2".Pressurep1p2[22])
      Move(in := "P3", out1 => "P3P4".Pressure34[16])
   END_RUNG
   RUNG wire#w1
      Move(in := "P4", out1 => "P3P4".Pressure34[22])
      Move(in := "Torque", out1 => "TS".TS[16])
      Move(in := "RPM", out1 => "TS".TS[22])
   END_RUNG
   RUNG wire#w1
      Move(in := "vibration", out1 => "Vib".vibration[10])
      Move(in := "VS", out1 => "VSVD".VsVd[16])
      Move(in := "Vd", out1 => "VSVD".VsVd[22])
   END_RUNG
   // the same network as SCL:
   IF "record1" AND "raw11" THEN
       "P1P2".Pressurep1p2[16] := "Suction_press";
       "P1P2".Pressurep1p2[22] := "Discharge_Press";
       "P3P4".Pressure34[16] := "P3";
       "P3P4".Pressure34[22] := "P4";
       "TS".TS[16] := "Torque";
       "TS".TS[22] := "RPM";
       "Vib".vibration[10] := "vibration";
       "VSVD".VsVd[16] := "VS";
       "VSVD".VsVd[22] := "Vd";
   END_IF;
END_REGION

REGION Network 15
   RUNG wire#powerrail
      Contact( "record1" )
      Contact( "raw11" )
      wire#w1
      Move(in := "Q", out1 => "QH".QH[16])
      Move(in := "H", out1 => "QH".QH[22])
      Move(in := "Shaft_power", out1 => "shftP.Pars".shaftP[16])
   END_RUNG
   RUNG wire#w1
      Move(in := "SP_ARS", out1 => "shftP.Pars".shaftP[22])
      Move(in := "QARS", out1 => "QarsHars".QarsHars[16])
      Move(in := "H_ARS", out1 => "QarsHars".QarsHars[22])
   END_RUNG
   RUNG wire#w1
      Move(in := "Efficiency", out1 => "EFF.NPSH"."EFF.NPSH"[16])
      Move(in := "Npsh", out1 => "EFF.NPSH"."EFF.NPSH"[22])
   END_RUNG
   // the same network as SCL:
   IF "record1" AND "raw11" THEN
       "QH".QH[16] := "Q";
       "QH".QH[22] := "H";
       "shftP.Pars".shaftP[16] := "Shaft_power";
       "shftP.Pars".shaftP[22] := "SP_ARS";
       "QarsHars".QarsHars[16] := "QARS";
       "QarsHars".QarsHars[22] := "H_ARS";
       "EFF.NPSH"."EFF.NPSH"[16] := "Efficiency";
       "EFF.NPSH"."EFF.NPSH"[22] := "Npsh";
   END_IF;
END_REGION

REGION Network 17
   RUNG wire#powerrail
      Contact( "record1" )
      Contact( "raw12" )
      wire#w1
      Move(in := "Suction_press", out1 => "P1P2".Pressurep1p2[17])
      Move(in := "Discharge_Press", out1 => "P1P2".Pressurep1p2[23])
      Move(in := "P3", out1 => "P3P4".Pressure34[17])
   END_RUNG
   RUNG wire#w1
      Move(in := "P4", out1 => "P3P4".Pressure34[23])
      Move(in := "Torque", out1 => "TS".TS[17])
      Move(in := "RPM", out1 => "TS".TS[23])
   END_RUNG
   RUNG wire#w1
      Move(in := "vibration", out1 => "Vib".vibration[11])
      Move(in := "VS", out1 => "VSVD".VsVd[17])
      Move(in := "Vd", out1 => "VSVD".VsVd[23])
   END_RUNG
   // the same network as SCL:
   IF "record1" AND "raw12" THEN
       "P1P2".Pressurep1p2[17] := "Suction_press";
       "P1P2".Pressurep1p2[23] := "Discharge_Press";
       "P3P4".Pressure34[17] := "P3";
       "P3P4".Pressure34[23] := "P4";
       "TS".TS[17] := "Torque";
       "TS".TS[23] := "RPM";
       "Vib".vibration[11] := "vibration";
       "VSVD".VsVd[17] := "VS";
       "VSVD".VsVd[23] := "Vd";
   END_IF;
END_REGION

REGION Network 18
   RUNG wire#powerrail
      Contact( "record" )
      Contact( "raw12" )
      wire#w1
      Move(in := "Q", out1 => "QH".QH[17])
      Move(in := "H", out1 => "QH".QH[23])
      Move(in := "Shaft_power", out1 => "shftP.Pars".shaftP[17])
   END_RUNG
   RUNG wire#w1
      Move(in := "SP_ARS", out1 => "shftP.Pars".shaftP[23])
      Move(in := "QARS", out1 => "QarsHars".QarsHars[17])
      Move(in := "H_ARS", out1 => "QarsHars".QarsHars[23])
   END_RUNG
   RUNG wire#w1
      Move(in := "Efficiency", out1 => "EFF.NPSH"."EFF.NPSH"[17])
      Move(in := "Npsh", out1 => "EFF.NPSH"."EFF.NPSH"[23])
   END_RUNG
   // the same network as SCL:
   IF "record" AND "raw12" THEN
       "QH".QH[17] := "Q";
       "QH".QH[23] := "H";
       "shftP.Pars".shaftP[17] := "Shaft_power";
       "shftP.Pars".shaftP[23] := "SP_ARS";
       "QarsHars".QarsHars[17] := "QARS";
       "QarsHars".QarsHars[23] := "H_ARS";
       "EFF.NPSH"."EFF.NPSH"[17] := "Efficiency";
       "EFF.NPSH"."EFF.NPSH"[23] := "Npsh";
   END_IF;
END_REGION
END_FUNCTION

ORGANIZATION_BLOCK "Main"   // OB1, LAD, ProgramCycle
TITLE = "Main Program Sweep (Cycle)"
{ S7_Optimized_Access := 'TRUE' }
VERSION : 0.1
   VAR_INPUT
      Initial_Call : Bool;   // Initial call of this OB
      Remanence : Bool;   // =True, if remanent data are available
   END_VAR
   VAR_TEMP   // added for the SCL form of the ladder/FBD networks
      _w1 : Bool;
      _w2 : Bool;
   END_VAR
BEGIN

REGION Network 2
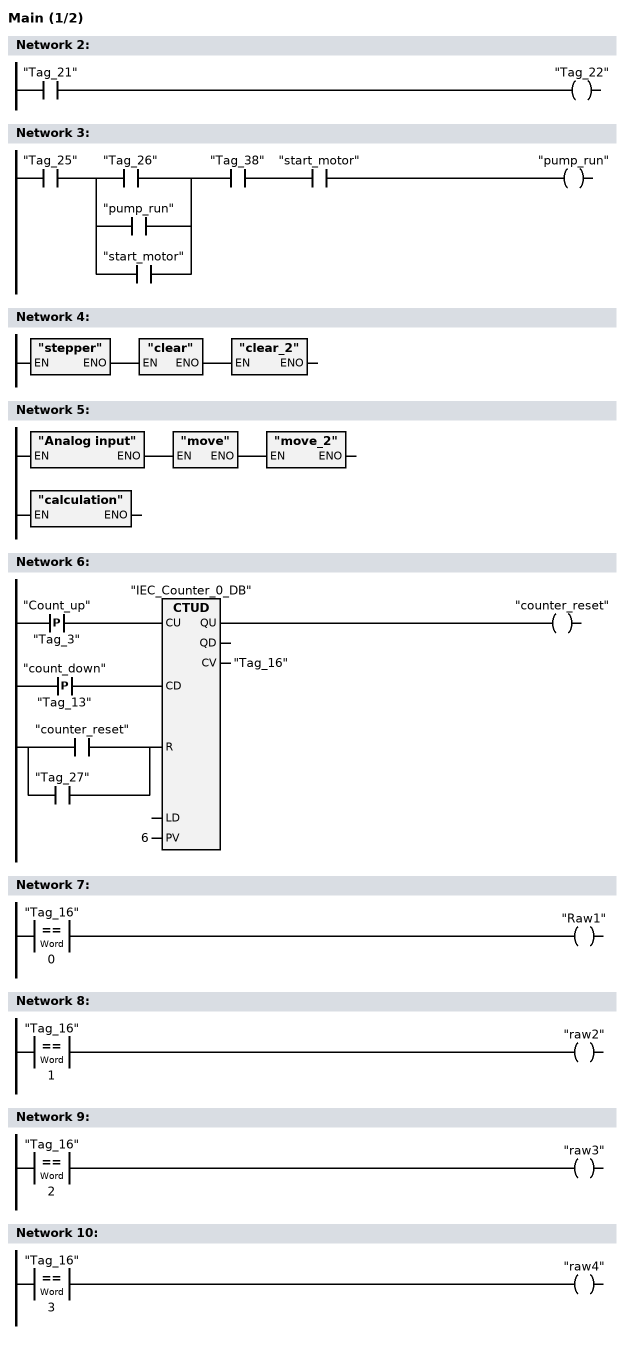
   RUNG wire#powerrail
      Contact( "Tag_21" )
      Coil( "Tag_22" )
   END_RUNG
   // the same network as SCL:
   "Tag_22" := "Tag_21";
END_REGION

REGION Network 3
   RUNG wire#powerrail
      Contact( "Tag_25" )
      wire#w1
      Contact( "Tag_26" )
      wire#w2
      Contact( "Tag_38" )
      Contact( "start_motor" )
      Coil( "pump_run" )
   END_RUNG
   RUNG wire#w1
      Contact( "pump_run" )
   END_RUNG wire#w2
   RUNG wire#w1
      Contact( "start_motor" )
   END_RUNG wire#w2
   // the same network as SCL:
   "pump_run" := "Tag_25" AND ("Tag_26" OR "pump_run" OR "start_motor") AND "Tag_38" AND "start_motor";
END_REGION

REGION Network 4
   RUNG wire#powerrail
      "stepper"()
      "clear"()
      "clear_2"()
   END_RUNG
   // the same network as SCL:
   "stepper"(ENO => #_w1);
   "clear"(EN := #_w1, ENO => #_w2);
   IF #_w2 THEN "clear_2"(); END_IF;
END_REGION

REGION Network 5
   RUNG wire#powerrail
      "Analog input"()
      "move"()
      "move_2"()
   END_RUNG
   RUNG wire#powerrail
      "calculation"()
   END_RUNG
   // the same network as SCL:
   "Analog input"(ENO => #_w1);
   "move"(EN := #_w1, ENO => #_w2);
   IF #_w2 THEN "move_2"(); END_IF;
   "calculation"();
END_REGION

REGION Network 6
   #_w1 := "Count_up" AND NOT "Tag_3";   // rising edge of "Count_up"
   "Tag_3" := "Count_up";
   #_w2 := "count_down" AND NOT "Tag_13";   // rising edge of "count_down"
   "Tag_13" := "count_down";
   "IEC_Counter_0_DB".CTUD(CU := #_w1, CD := #_w2, R := "counter_reset" OR "Tag_27", PV := 6, CV => "Tag_16");
   "counter_reset" := "IEC_Counter_0_DB".QU;
END_REGION

REGION Network 7
   RUNG wire#powerrail
      { S7_Templates := "SrcType := Word" } EQ_Contact(in1 := "Tag_16", in2 := 0)
      Coil( "Raw1" )
   END_RUNG
   // the same network as SCL:
   "Raw1" := "Tag_16" = 0;
END_REGION

REGION Network 8
   RUNG wire#powerrail
      { S7_Templates := "SrcType := Word" } EQ_Contact(in1 := "Tag_16", in2 := 1)
      Coil( "raw2" )
   END_RUNG
   // the same network as SCL:
   "raw2" := "Tag_16" = 1;
END_REGION

REGION Network 9
   RUNG wire#powerrail
      { S7_Templates := "SrcType := Word" } EQ_Contact(in1 := "Tag_16", in2 := 2)
      Coil( "raw3" )
   END_RUNG
   // the same network as SCL:
   "raw3" := "Tag_16" = 2;
END_REGION

REGION Network 10
   RUNG wire#powerrail
      { S7_Templates := "SrcType := Word" } EQ_Contact(in1 := "Tag_16", in2 := 3)
      Coil( "raw4" )
   END_RUNG
   // the same network as SCL:
   "raw4" := "Tag_16" = 3;
END_REGION

REGION Network 11
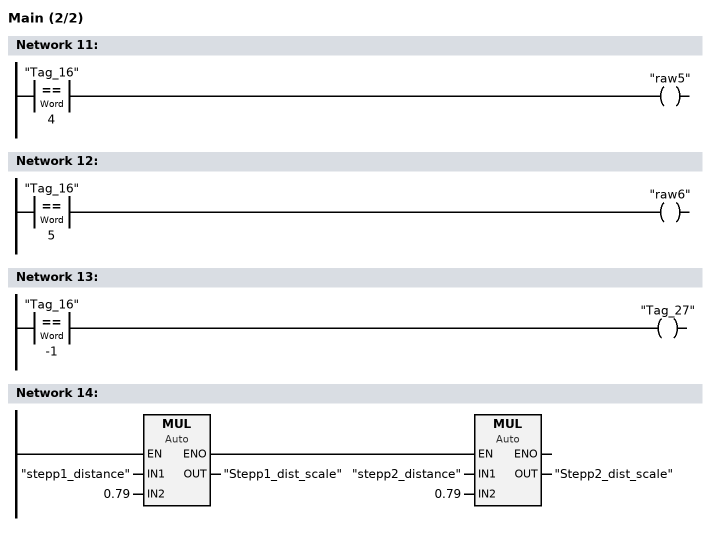
   RUNG wire#powerrail
      { S7_Templates := "SrcType := Word" } EQ_Contact(in1 := "Tag_16", in2 := 4)
      Coil( "raw5" )
   END_RUNG
   // the same network as SCL:
   "raw5" := "Tag_16" = 4;
END_REGION

REGION Network 12
   RUNG wire#powerrail
      { S7_Templates := "SrcType := Word" } EQ_Contact(in1 := "Tag_16", in2 := 5)
      Coil( "raw6" )
   END_RUNG
   // the same network as SCL:
   "raw6" := "Tag_16" = 5;
END_REGION

REGION Network 13
   RUNG wire#powerrail
      { S7_Templates := "SrcType := Word" } EQ_Contact(in1 := "Tag_16", in2 := -1)
      Coil( "Tag_27" )
   END_RUNG
   // the same network as SCL:
   "Tag_27" := "Tag_16" = (-1);
END_REGION

REGION Network 14
   RUNG wire#powerrail
      Mul(in1 := "stepp1_distance", in2 := 0.79, out => "Stepp1_dist_scale")
      Mul(in1 := "stepp2_distance", in2 := 0.79, out => "Stepp2_dist_scale")
   END_RUNG
   // the same network as SCL:
   "Stepp1_dist_scale" := "stepp1_distance" * 0.79;
   "Stepp2_dist_scale" := "stepp2_distance" * 0.79;
END_REGION
END_ORGANIZATION_BLOCK

(* ===== HMI "HMI_RT_1" =====
system functions are stored by id; their names below are inferred from use
connection "HMI_Connection_1": ETHERNET, S7_1200_OMS

HMI tags "Default tag table"
   "Tag_33" : Real = PLC vibration AT %MD100, 1 s
   "Tag_11" : Bool = PLC Tag_11 AT %M20.0, 1 s
   "Tag_9" : Real = PLC P3 AT %MD60, 1 s
   "Tag_9(1)" : Bool = PLC Tag_9 AT %M20.1, 1 s
   "compare" : Real = PLC compare AT %MD104, 1 s
   "Referance_motor_speed" : Real = PLC Referance_motor_speed AT %MD176, 1 s
   "RPM" : Real = PLC RPM AT %MD92, 1 s
   "Raw1" : Bool = PLC Raw1 AT %M30.3, 1 s
   "raw2" : Bool = PLC raw2 AT %M30.4, 1 s
   "raw3" : Bool = PLC raw3 AT %M30.5, 1 s
   "raw4" : Bool = PLC raw4 AT %M30.6, 1 s
   "raw5" : Bool = PLC raw5 AT %M30.7, 1 s
   "raw6" : Bool = PLC raw6 AT %M31.4, 1 s
   "Count_up" : Bool = PLC Count_up AT %M30.0, 1 s
   "count_down" : Bool = PLC count_down AT %M30.1, 1 s
   "Suction_press" : Real = PLC Suction_press AT %MD44, 1 s
   "Discharge_Press" : Real = PLC Discharge_Press AT %MD52, 1 s
   "P4" : Real = PLC P4 AT %MD68, 1 s
   "Torque" : Real = PLC Torque AT %MD84, 1 s
   "VS" : Real = PLC VS AT %MD152, 1 s
   "Vd" : Real = PLC Vd AT %MD156, 1 s
   "Q" : Real = PLC Q AT %MD148, 1 s
   "H" : Real = PLC H AT %MD168, 1 s
   "Shaft_power" : Real = PLC Shaft_power AT %MD172, 1 s
   "QARS" : Real = PLC QARS AT %MD180, 1 s
   "H_ARS" : Real = PLC H_ARS AT %MD200, 1 s
   "Efficiency" : Real = PLC Efficiency AT %MD208, 1 s
   "Npsh" : Real = PLC Npsh AT %MD212, 1 s
   "P1P2_Pressurep1p2{0}" : Real = PLC P1P2.Pressurep1p2[0], 1 s
   "P1P2_Pressurep1p2{1}" : Real = PLC P1P2.Pressurep1p2[1], 1 s
   "P1P2_Pressurep1p2{2}" : Real = PLC P1P2.Pressurep1p2[2], 1 s
   "P1P2_Pressurep1p2{3}" : Real = PLC P1P2.Pressurep1p2[3], 1 s
   "P1P2_Pressurep1p2{4}" : Real = PLC P1P2.Pressurep1p2[4], 1 s
   "P1P2_Pressurep1p2{5}" : Real = PLC P1P2.Pressurep1p2[5], 1 s
   "P1P2_Pressurep1p2{6}" : Real = PLC P1P2.Pressurep1p2[6], 1 s
   "P1P2_Pressurep1p2{7}" : Real = PLC P1P2.Pressurep1p2[7], 1 s
   "P1P2_Pressurep1p2{8}" : Real = PLC P1P2.Pressurep1p2[8], 1 s
   "P1P2_Pressurep1p2{9}" : Real = PLC P1P2.Pressurep1p2[9], 1 s
   "P1P2_Pressurep1p2{10}" : Real = PLC P1P2.Pressurep1p2[10], 1 s
   "P1P2_Pressurep1p2{11}" : Real = PLC P1P2.Pressurep1p2[11], 1 s
   "P3P4_Pressure34{0}" : Real = PLC P3P4.Pressure34[0], 1 s
   "P3P4_Pressure34{1}" : Real = PLC P3P4.Pressure34[1], 1 s
   "P3P4_Pressure34{2}" : Real = PLC P3P4.Pressure34[2], 1 s
   "P3P4_Pressure34{3}" : Real = PLC P3P4.Pressure34[3], 1 s
   "P3P4_Pressure34{4}" : Real = PLC P3P4.Pressure34[4], 1 s
   "P3P4_Pressure34{5}" : Real = PLC P3P4.Pressure34[5], 1 s
   "P3P4_Pressure34{6}" : Real = PLC P3P4.Pressure34[6], 1 s
   "P3P4_Pressure34{7}" : Real = PLC P3P4.Pressure34[7], 1 s
   "P3P4_Pressure34{8}" : Real = PLC P3P4.Pressure34[8], 1 s
   "P3P4_Pressure34{9}" : Real = PLC P3P4.Pressure34[9], 1 s
   "P3P4_Pressure34{10}" : Real = PLC P3P4.Pressure34[10], 1 s
   "P3P4_Pressure34{11}" : Real = PLC P3P4.Pressure34[11], 1 s
   "TS_TS{0}" : Real = PLC TS.TS[0], 1 s
   "TS_TS{1}" : Real = PLC TS.TS[1], 1 s
   "TS_TS{2}" : Real = PLC TS.TS[2], 1 s
   "TS_TS{3}" : Real = PLC TS.TS[3], 1 s
   "TS_TS{4}" : Real = PLC TS.TS[4], 1 s
   "TS_TS{5}" : Real = PLC TS.TS[5], 1 s
   "TS_TS{6}" : Real = PLC TS.TS[6], 1 s
   "TS_TS{7}" : Real = PLC TS.TS[7], 1 s
   "TS_TS{8}" : Real = PLC TS.TS[8], 1 s
   "TS_TS{9}" : Real = PLC TS.TS[9], 1 s
   "TS_TS{10}" : Real = PLC TS.TS[10], 1 s
   "TS_TS{11}" : Real = PLC TS.TS[11], 1 s
   "Vib_vibration{0}" : Real = PLC Vib.vibration[0], 1 s
   "Vib_vibration{1}" : Real = PLC Vib.vibration[1], 1 s
   "Vib_vibration{2}" : Real = PLC Vib.vibration[2], 1 s
   "Vib_vibration{3}" : Real = PLC Vib.vibration[3], 1 s
   "Vib_vibration{4}" : Real = PLC Vib.vibration[4], 1 s
   "Vib_vibration{5}" : Real = PLC Vib.vibration[5], 1 s
   "VSVD_VsVd{0}" : Real = PLC VSVD.VsVd[0], 1 s
   "VSVD_VsVd{1}" : Real = PLC VSVD.VsVd[1], 1 s
   "VSVD_VsVd{2}" : Real = PLC VSVD.VsVd[2], 1 s
   "VSVD_VsVd{3}" : Real = PLC VSVD.VsVd[3], 1 s
   "VSVD_VsVd{4}" : Real = PLC VSVD.VsVd[4], 1 s
   "VSVD_VsVd{5}" : Real = PLC VSVD.VsVd[5], 1 s
   "VSVD_VsVd{6}" : Real = PLC VSVD.VsVd[6], 1 s
   "VSVD_VsVd{7}" : Real = PLC VSVD.VsVd[7], 1 s
   "VSVD_VsVd{8}" : Real = PLC VSVD.VsVd[8], 1 s
   "VSVD_VsVd{9}" : Real = PLC VSVD.VsVd[9], 1 s
   "VSVD_VsVd{10}" : Real = PLC VSVD.VsVd[10], 1 s
   "VSVD_VsVd{11}" : Real = PLC VSVD.VsVd[11], 1 s
   "QH_QH{0}" : Real = PLC QH.QH[0], 1 s
   "QH_QH{1}" : Real = PLC QH.QH[1], 1 s
   "QH_QH{2}" : Real = PLC QH.QH[2], 1 s
   "QH_QH{3}" : Real = PLC QH.QH[3], 1 s
   "QH_QH{4}" : Real = PLC QH.QH[4], 1 s
   "QH_QH{5}" : Real = PLC QH.QH[5], 1 s
   "QH_QH{6}" : Real = PLC QH.QH[6], 1 s
   "QH_QH{7}" : Real = PLC QH.QH[7], 1 s
   "QH_QH{8}" : Real = PLC QH.QH[8], 1 s
   "QH_QH{9}" : Real = PLC QH.QH[9], 1 s
   "QH_QH{10}" : Real = PLC QH.QH[10], 1 s
   "QH_QH{11}" : Real = PLC QH.QH[11], 1 s
   "shftP.Pars_shaftP{0}" : Real = PLC "shftP.Pars".shaftP[0], 1 s
   "shftP.Pars_shaftP{1}" : Real = PLC "shftP.Pars".shaftP[1], 1 s
   "shftP.Pars_shaftP{2}" : Real = PLC "shftP.Pars".shaftP[2], 1 s
   "shftP.Pars_shaftP{3}" : Real = PLC "shftP.Pars".shaftP[3], 1 s
   "shftP.Pars_shaftP{4}" : Real = PLC "shftP.Pars".shaftP[4], 1 s
   "shftP.Pars_shaftP{5}" : Real = PLC "shftP.Pars".shaftP[5], 1 s
   "shftP.Pars_shaftP{6}" : Real = PLC "shftP.Pars".shaftP[6], 1 s
   "shftP.Pars_shaftP{7}" : Real = PLC "shftP.Pars".shaftP[7], 1 s
   "shftP.Pars_shaftP{8}" : Real = PLC "shftP.Pars".shaftP[8], 1 s
   "shftP.Pars_shaftP{9}" : Real = PLC "shftP.Pars".shaftP[9], 1 s
   "shftP.Pars_shaftP{10}" : Real = PLC "shftP.Pars".shaftP[10], 1 s
   "shftP.Pars_shaftP{11}" : Real = PLC "shftP.Pars".shaftP[11], 1 s
   "QarsHars_QarsHars{0}" : Real = PLC QarsHars.QarsHars[0], 1 s
   "QarsHars_QarsHars{1}" : Real = PLC QarsHars.QarsHars[1], 1 s
   "QarsHars_QarsHars{2}" : Real = PLC QarsHars.QarsHars[2], 1 s
   "QarsHars_QarsHars{3}" : Real = PLC QarsHars.QarsHars[3], 1 s
   "QarsHars_QarsHars{4}" : Real = PLC QarsHars.QarsHars[4], 1 s
   "QarsHars_QarsHars{5}" : Real = PLC QarsHars.QarsHars[5], 1 s
   "QarsHars_QarsHars{6}" : Real = PLC QarsHars.QarsHars[6], 1 s
   "QarsHars_QarsHars{7}" : Real = PLC QarsHars.QarsHars[7], 1 s
   "QarsHars_QarsHars{8}" : Real = PLC QarsHars.QarsHars[8], 1 s
   "QarsHars_QarsHars{9}" : Real = PLC QarsHars.QarsHars[9], 1 s
   "QarsHars_QarsHars{10}" : Real = PLC QarsHars.QarsHars[10], 1 s
   "QarsHars_QarsHars{11}" : Real = PLC QarsHars.QarsHars[11], 1 s
   "EFF.NPSH_EFF.NPSH{0}" : Real = PLC "EFF.NPSH"."EFF.NPSH"[0], 1 s
   "EFF.NPSH_EFF.NPSH{1}" : Real = PLC "EFF.NPSH"."EFF.NPSH"[1], 1 s
   "EFF.NPSH_EFF.NPSH{2}" : Real = PLC "EFF.NPSH"."EFF.NPSH"[2], 1 s
   "EFF.NPSH_EFF.NPSH{3}" : Real = PLC "EFF.NPSH"."EFF.NPSH"[3], 1 s
   "EFF.NPSH_EFF.NPSH{4}" : Real = PLC "EFF.NPSH"."EFF.NPSH"[4], 1 s
   "EFF.NPSH_EFF.NPSH{5}" : Real = PLC "EFF.NPSH"."EFF.NPSH"[5], 1 s
   "EFF.NPSH_EFF.NPSH{6}" : Real = PLC "EFF.NPSH"."EFF.NPSH"[6], 1 s
   "EFF.NPSH_EFF.NPSH{7}" : Real = PLC "EFF.NPSH"."EFF.NPSH"[7], 1 s
   "EFF.NPSH_EFF.NPSH{12}" : Real = PLC "EFF.NPSH"."EFF.NPSH"[12], 1 s
   "EFF.NPSH_EFF.NPSH{13}" : Real = PLC "EFF.NPSH"."EFF.NPSH"[13], 1 s
   "SP_ARS" : Real = PLC SP_ARS AT %MD204, 1 s
   "pump_run" : Bool = PLC pump_run AT %Q0.6, 1 s
   "EFF.NPSH_EFF.NPSH{8}" : Real = PLC "EFF.NPSH"."EFF.NPSH"[8], 1 s
   "EFF.NPSH_EFF.NPSH{9}" : Real = PLC "EFF.NPSH"."EFF.NPSH"[9], 1 s
   "EFF.NPSH_EFF.NPSH{10}" : Real = PLC "EFF.NPSH"."EFF.NPSH"[10], 1 s
   "EFF.NPSH_EFF.NPSH{11}" : Real = PLC "EFF.NPSH"."EFF.NPSH"[11], 1 s
   "record" : Bool = PLC record AT %M31.5, 1 s
   "start_motor" : Bool = PLC start_motor AT %M32.2, 1 s
   "clear All" : Bool = PLC "clear All" AT %M32.3, 1 s
   "stepp1_distance" : Real = PLC stepp1_distance AT %MD216, 1 s
   "Axis_1_Direction" : Bool = PLC Axis_1_Direction AT %Q0.1, 1 s
   "stepp1_start" : Bool = PLC stepp1_start AT %M31.7, 1 s
   "Temperature" : Real = PLC Temperature AT %MD76, 1 s
   "stepp1_enab" : Bool = PLC stepp1_enab AT %M31.6, 1 s
   "stepp1_home" : Bool = PLC stepp1_home AT %M32.5, 1 s
   "stepp2_enab" : Bool = PLC stepp2_enab AT %M32.7, 1 s
   "stepp2_home" : Bool = PLC stepp2_home AT %M32.6, 1 s
   "stepp2_excut" : Bool = PLC stepp2_excut AT %M33.0, 1 s
   "stepp2_distance" : Real = PLC stepp2_distance AT %MD220, 1 s
   "configuration" : WChar = PLC configuration AT %MW232, 1 s
   "date" : Date = PLC date AT %MW234, 1 s
   "time" : Time_Of_Day = PLC time AT %MD236, 1 s
   "time_1" : Time_Of_Day = PLC time_1 AT %MD240, 1 s
   "P3P4_Pressure34{0}(1)" : Real = PLC P3P4.Pressure34[12] AT %DB1.DBD0, 1 s
   "P3P4_Pressure34{1}(1)" : Real = PLC P3P4.Pressure34[13] AT %DB1.DBD0, 1 s
   "P3P4_Pressure34{2}(1)" : Real = PLC P3P4.Pressure34[14] AT %DB1.DBD0, 1 s
   "P3P4_Pressure34{3}(1)" : Real = PLC P3P4.Pressure34[15] AT %DB1.DBD0, 1 s
   "P3P4_Pressure34{4}(1)" : Real = PLC P3P4.Pressure34[16] AT %DB1.DBD0, 1 s
   "P3P4_Pressure34{5}(1)" : Real = PLC P3P4.Pressure34[17] AT %DB1.DBD0, 1 s
   "P3P4_Pressure34{6}(1)" : Real = PLC P3P4.Pressure34[18] AT %DB1.DBD0, 1 s
   "P3P4_Pressure34{7}(1)" : Real = PLC P3P4.Pressure34[19] AT %DB1.DBD0, 1 s
   "P3P4_Pressure34{8}(1)" : Real = PLC P3P4.Pressure34[20] AT %DB1.DBD0, 1 s
   "P3P4_Pressure34{9}(1)" : Real = PLC P3P4.Pressure34[21] AT %DB1.DBD0, 1 s
   "P3P4_Pressure34{10}(1)" : Real = PLC P3P4.Pressure34[22] AT %DB1.DBD0, 1 s
   "P3P4_Pressure34{11}(1)" : Real = PLC P3P4.Pressure34[23] AT %DB1.DBD0, 1 s
   "P1P2_Pressurep1p2{0}(1)" : Real = PLC P1P2.Pressurep1p2[12] AT %DB1.DBD0, 1 s
   "P1P2_Pressurep1p2{0}(2)" : Real = PLC P1P2.Pressurep1p2[13] AT %DB1.DBD0, 1 s
   "P1P2_Pressurep1p2{0}(3)" : Real = PLC P1P2.Pressurep1p2[14] AT %DB1.DBD0, 1 s
   "P1P2_Pressurep1p2{0}(4)" : Real = PLC P1P2.Pressurep1p2[15] AT %DB1.DBD0, 1 s
   "P1P2_Pressurep1p2{0}(5)" : Real = PLC P1P2.Pressurep1p2[16] AT %DB1.DBD0, 1 s
   "P1P2_Pressurep1p2{0}(6)" : Real = PLC P1P2.Pressurep1p2[17] AT %DB1.DBD0, 1 s
   "P1P2_Pressurep1p2{0}(7)" : Real = PLC P1P2.Pressurep1p2[18] AT %DB1.DBD0, 1 s
   "P1P2_Pressurep1p2{0}(8)" : Real = PLC P1P2.Pressurep1p2[19] AT %DB1.DBD0, 1 s
   "P1P2_Pressurep1p2{0}(9)" : Real = PLC P1P2.Pressurep1p2[20] AT %DB1.DBD0, 1 s
   "P1P2_Pressurep1p2{0}(10)" : Real = PLC P1P2.Pressurep1p2[21] AT %DB1.DBD0, 1 s
   "P1P2_Pressurep1p2{0}(11)" : Real = PLC P1P2.Pressurep1p2[22] AT %DB1.DBD0, 1 s
   "P1P2_Pressurep1p2{0}(12)" : Real = PLC P1P2.Pressurep1p2[23] AT %DB1.DBD0, 1 s
   "TS_TS{0}(1)" : Real = PLC TS.TS[12] AT %DB1.DBD0, 1 s
   "TS_TS{1}(1)" : Real = PLC TS.TS[13] AT %DB1.DBD0, 1 s
   "TS_TS{2}(1)" : Real = PLC TS.TS[14] AT %DB1.DBD0, 1 s
   "TS_TS{3}(1)" : Real = PLC TS.TS[15] AT %DB1.DBD0, 1 s
   "TS_TS{4}(1)" : Real = PLC TS.TS[16] AT %DB1.DBD0, 1 s
   "TS_TS{5}(1)" : Real = PLC TS.TS[17] AT %DB1.DBD0, 1 s
   "TS_TS{6}(1)" : Real = PLC TS.TS[18] AT %DB1.DBD0, 1 s
   "TS_TS{7}(1)" : Real = PLC TS.TS[19] AT %DB1.DBD0, 1 s
   "TS_TS{8}(1)" : Real = PLC TS.TS[20] AT %DB1.DBD0, 1 s
   "TS_TS{9}(1)" : Real = PLC TS.TS[21] AT %DB1.DBD0, 1 s
   "TS_TS{10}(1)" : Real = PLC TS.TS[22] AT %DB1.DBD0, 1 s
   "TS_TS{11}(1)" : Real = PLC TS.TS[23] AT %DB1.DBD0, 1 s
   "Vib_vibration{0}(1)" : Real = PLC Vib.vibration[6] AT %DB1.DBD0, 1 s
   "Vib_vibration{1}(1)" : Real = PLC Vib.vibration[7] AT %DB1.DBD0, 1 s
   "Vib_vibration{2}(1)" : Real = PLC Vib.vibration[8] AT %DB1.DBD0, 1 s
   "Vib_vibration{3}(1)" : Real = PLC Vib.vibration[9] AT %DB1.DBD0, 1 s
   "Vib_vibration{4}(1)" : Real = PLC Vib.vibration[10] AT %DB1.DBD0, 1 s
   "Vib_vibration{5}(1)" : Real = PLC Vib.vibration[11] AT %DB1.DBD0, 1 s
   "VSVD_VsVd{0}(1)" : Real = PLC VSVD.VsVd[12] AT %DB1.DBD0, 1 s
   "VSVD_VsVd{1}(1)" : Real = PLC VSVD.VsVd[13] AT %DB1.DBD0, 1 s
   "VSVD_VsVd{2}(1)" : Real = PLC VSVD.VsVd[14] AT %DB1.DBD0, 1 s
   "VSVD_VsVd{3}(1)" : Real = PLC VSVD.VsVd[15] AT %DB1.DBD0, 1 s
   "VSVD_VsVd{4}(1)" : Real = PLC VSVD.VsVd[16] AT %DB1.DBD0, 1 s
   "VSVD_VsVd{5}(1)" : Real = PLC VSVD.VsVd[17] AT %DB1.DBD0, 1 s
   "VSVD_VsVd{6}(1)" : Real = PLC VSVD.VsVd[18] AT %DB1.DBD0, 1 s
   "VSVD_VsVd{7}(1)" : Real = PLC VSVD.VsVd[19] AT %DB1.DBD0, 1 s
   "VSVD_VsVd{8}(1)" : Real = PLC VSVD.VsVd[20] AT %DB1.DBD0, 1 s
   "VSVD_VsVd{9}(1)" : Real = PLC VSVD.VsVd[21] AT %DB1.DBD0, 1 s
   "VSVD_VsVd{10}(1)" : Real = PLC VSVD.VsVd[22] AT %DB1.DBD0, 1 s
   "VSVD_VsVd{11}(1)" : Real = PLC VSVD.VsVd[23] AT %DB1.DBD0, 1 s
   "shftP.Pars_shaftP{0}(1)" : Real = PLC "shftP.Pars".shaftP[12] AT %DB1.DBD0, 1 s
   "shftP.Pars_shaftP{1}(1)" : Real = PLC "shftP.Pars".shaftP[13] AT %DB1.DBD0, 1 s
   "shftP.Pars_shaftP{2}(1)" : Real = PLC "shftP.Pars".shaftP[14] AT %DB1.DBD0, 1 s
   "shftP.Pars_shaftP{3}(1)" : Real = PLC "shftP.Pars".shaftP[15] AT %DB1.DBD0, 1 s
   "shftP.Pars_shaftP{4}(1)" : Real = PLC "shftP.Pars".shaftP[16] AT %DB1.DBD0, 1 s
   "shftP.Pars_shaftP{5}(1)" : Real = PLC "shftP.Pars".shaftP[17] AT %DB1.DBD0, 1 s
   "shftP.Pars_shaftP{6}(1)" : Real = PLC "shftP.Pars".shaftP[18] AT %DB1.DBD0, 1 s
   "shftP.Pars_shaftP{7}(1)" : Real = PLC "shftP.Pars".shaftP[19] AT %DB1.DBD0, 1 s
   "shftP.Pars_shaftP{8}(1)" : Real = PLC "shftP.Pars".shaftP[20] AT %DB1.DBD0, 1 s
   "shftP.Pars_shaftP{9}(1)" : Real = PLC "shftP.Pars".shaftP[21] AT %DB1.DBD0, 1 s
   "shftP.Pars_shaftP{10}(1)" : Real = PLC "shftP.Pars".shaftP[22] AT %DB1.DBD0, 1 s
   "shftP.Pars_shaftP{11}(1)" : Real = PLC "shftP.Pars".shaftP[23] AT %DB1.DBD0, 1 s
   "QarsHars_QarsHars{0}(1)" : Real = PLC QarsHars.QarsHars[12] AT %DB1.DBD0, 1 s
   "QarsHars_QarsHars{1}(1)" : Real = PLC QarsHars.QarsHars[13] AT %DB1.DBD0, 1 s
   "QarsHars_QarsHars{2}(1)" : Real = PLC QarsHars.QarsHars[14] AT %DB1.DBD0, 1 s
   "QarsHars_QarsHars{3}(1)" : Real = PLC QarsHars.QarsHars[15] AT %DB1.DBD0, 1 s
   "QarsHars_QarsHars{4}(1)" : Real = PLC QarsHars.QarsHars[16] AT %DB1.DBD0, 1 s
   "QarsHars_QarsHars{5}(1)" : Real = PLC QarsHars.QarsHars[17] AT %DB1.DBD0, 1 s
   "QarsHars_QarsHars{6}(1)" : Real = PLC QarsHars.QarsHars[18] AT %DB1.DBD0, 1 s
   "QarsHars_QarsHars{7}(1)" : Real = PLC QarsHars.QarsHars[19] AT %DB1.DBD0, 1 s
   "QarsHars_QarsHars{8}(1)" : Real = PLC QarsHars.QarsHars[20] AT %DB1.DBD0, 1 s
   "QarsHars_QarsHars{9}(1)" : Real = PLC QarsHars.QarsHars[21] AT %DB1.DBD0, 1 s
   "QarsHars_QarsHars{10}(1)" : Real = PLC QarsHars.QarsHars[22] AT %DB1.DBD0, 1 s
   "QarsHars_QarsHars{11}(1)" : Real = PLC QarsHars.QarsHars[23] AT %DB1.DBD0, 1 s
   "QH_QH{0}(1)" : Real = PLC QH.QH[12] AT %DB1.DBD0, 1 s
   "QH_QH{1}(1)" : Real = PLC QH.QH[13] AT %DB1.DBD0, 1 s
   "QH_QH{2}(1)" : Real = PLC QH.QH[14] AT %DB1.DBD0, 1 s
   "QH_QH{4}(1)" : Real = PLC QH.QH[16] AT %DB1.DBD0, 1 s
   "QH_QH{3}(1)" : Real = PLC QH.QH[15] AT %DB1.DBD0, 1 s
   "QH_QH{5}(1)" : Real = PLC QH.QH[17] AT %DB1.DBD0, 1 s
   "QH_QH{6}(1)" : Real = PLC QH.QH[18] AT %DB1.DBD0, 1 s
   "QH_QH{7}(1)" : Real = PLC QH.QH[19] AT %DB1.DBD0, 1 s
   "QH_QH{8}(1)" : Real = PLC QH.QH[20] AT %DB1.DBD0, 1 s
   "QH_QH{9}(1)" : Real = PLC QH.QH[21] AT %DB1.DBD0, 1 s
   "QH_QH{10}(1)" : Real = PLC QH.QH[22] AT %DB1.DBD0, 1 s
   "QH_QH{11}(1)" : Real = PLC QH.QH[23] AT %DB1.DBD0, 1 s
   "EFF.NPSH_EFF.NPSH{0}(1)" : Real = PLC "EFF.NPSH"."EFF.NPSH"[12] AT %DB1.DBD0, 1 s
   "EFF.NPSH_EFF.NPSH{1}(1)" : Real = PLC "EFF.NPSH"."EFF.NPSH"[13] AT %DB1.DBD0, 1 s
   "EFF.NPSH_EFF.NPSH{2}(1)" : Real = PLC "EFF.NPSH"."EFF.NPSH"[14] AT %DB1.DBD0, 1 s
   "EFF.NPSH_EFF.NPSH{3}(1)" : Real = PLC "EFF.NPSH"."EFF.NPSH"[15] AT %DB1.DBD0, 1 s
   "EFF.NPSH_EFF.NPSH{4}(1)" : Real = PLC "EFF.NPSH"."EFF.NPSH"[16] AT %DB1.DBD0, 1 s
   "EFF.NPSH_EFF.NPSH{5}(1)" : Real = PLC "EFF.NPSH"."EFF.NPSH"[17] AT %DB1.DBD0, 1 s
   "EFF.NPSH_EFF.NPSH{6}(1)" : Real = PLC "EFF.NPSH"."EFF.NPSH"[18] AT %DB1.DBD0, 1 s
   "EFF.NPSH_EFF.NPSH{7}(1)" : Real = PLC "EFF.NPSH"."EFF.NPSH"[19] AT %DB1.DBD0, 1 s
   "EFF.NPSH_EFF.NPSH{8}(1)" : Real = PLC "EFF.NPSH"."EFF.NPSH"[20] AT %DB1.DBD0, 1 s
   "EFF.NPSH_EFF.NPSH{9}(1)" : Real = PLC "EFF.NPSH"."EFF.NPSH"[21] AT %DB1.DBD0, 1 s
   "EFF.NPSH_EFF.NPSH{10}(1)" : Real = PLC "EFF.NPSH"."EFF.NPSH"[22] AT %DB1.DBD0, 1 s
   "EFF.NPSH_EFF.NPSH{11}(1)" : Real = PLC "EFF.NPSH"."EFF.NPSH"[23] AT %DB1.DBD0, 1 s
   "deviation" : Real = PLC deviation AT %MD244, 1 s
   "deviation_1" : Real = PLC deviation_1.deviation_1 AT %DB1.DBD0, 1 s
   "deviation_2" : Real = PLC deviation_1.deviation_2 AT %DB1.DBD0, 1 s
   "deviation_3" : Real = PLC deviation_1.deviation_3 AT %DB1.DBD0, 1 s
   "deviation_4" : Real = PLC deviation_1.deviation_4 AT %DB1.DBD0, 1 s
   "deviation_5" : Real = PLC deviation_1.deviation_5 AT %DB1.DBD0, 1 s
   "deviation_0" : Real = PLC deviation_1.deviation_0 AT %DB1.DBD0, 1 s
   "raw7" : Bool = PLC raw7 AT %M33.1, 1 s
   "raw8" : Bool = PLC raw8 AT %M33.2, 1 s
   "raw9" : Bool = PLC raw9 AT %M33.3, 1 s
   "raw10" : Bool = PLC raw10 AT %M33.4, 1 s
   "raw11" : Bool = PLC raw11 AT %M33.5, 1 s
   "raw12" : Bool = PLC raw12 AT %M33.6, 1 s

screen "home" 1024x761
   GraphicView "Graphic view_8" at 788,526 size 43x76; Picture "d2bzw5qd.1cx_1"
   Button "Button_2" at 858,698 size 156x56; TextOff 'Exit'
      on Press: StopRuntime(0)
   GraphicView "Template_Graphic view_4" at 180,442 size 128x119; Picture "Graphic_11"
   GraphicView "Graphic view_3" at 832,376 size 49x107; Picture "Graphic_20"
   GraphicView "Graphic view_6" at 265,239 size 37x52; Picture "Graphic_24"
   GraphicView "Template_Graphic view_8" at 306,482 size 399x65; Picture "Graphic_17"
   GraphicView "Graphic view_11" at 831,481 size 49x65; Picture "Graphic_32"
   Rectangle "Rectangle_7" at 187,489 size 17x49
      Appearance <- "pump_run"
   IOField "I/O field_51" at 360,450 size 64x32; FormatPattern s99.99
      ProcessValue <- "Suction_press"
   IOField "I/O field_52" at 192,415 size 68x32; FormatPattern 99.99
      ProcessValue <- "Discharge_Press"
   TextField "Text field_14" at 422,455 size 45x20; Text 'bar'
   TextField "Text field_15" at 79,505 size 42x23; Text 'RPM'
   IOField "I/O field_49" at 124,501 size 53x32; FormatPattern 9999
      ProcessValue <- "RPM"
   GraphicView "Graphic view_4" at 795,134 size 122x247; Picture "Graphic_2"
   GraphicView "Graphic view_1" at 704,473 size 61x63; Picture "Graphic_3"
   GraphicView "Template_Graphic view_5" at 736,481 size 96x65; Picture "Graphic_17"
   GraphicView "Graphic view_7" at 265,288 size 35x159; Picture "Graphic_20"
   GraphicView "Template_Graphic view_13" at 301,240 size 179x50; Picture "Graphic_17"
   GraphicView "Template_Graphic view_14" at 591,191 size 59x97; Picture "Graphic_15"
   GraphicView "Graphic view_16" at 478,239 size 30x48; Picture "Graphic_5"
   GraphicView "Template_Graphic view_15" at 509,241 size 88x50; Picture "Graphic_17"
   GraphicView "Template_Graphic view_16" at 645,240 size 30x50; Picture "Graphic_17"
   GraphicView "Graphic view_17" at 675,239 size 38x52; Picture "Graphic_32"
   GraphicView "Graphic view_18" at 675,121 size 37x119; Picture "Graphic_20"
   GraphicView "Graphic view_19" at 675,70 size 37x52; Picture "Graphic_24"
   GraphicView "Template_Graphic view_3" at 713,70 size 115x50; Picture "Graphic_17"
   GraphicView "Graphic view_21" at 828,70 size 38x52; Picture "Graphic_30"
   GraphicView "Graphic view_22" at 828,70 size 37x52; Picture "Graphic_31"
      Visibility <- "pump_run"
   GraphicView "Template_Graphic view_17" at 711,71 size 117x50; Picture "Graphic_18"
      Visibility <- "pump_run"
   GraphicView "Graphic view_23" at 675,70 size 37x52; Picture "Graphic_34"
      Visibility <- "pump_run"
   GraphicView "Graphic view_24" at 675,120 size 37x122; Picture "Graphic_21"
      Visibility <- "pump_run"
   GraphicView "Graphic view_25" at 675,240 size 38x52; Picture "Graphic_33"
      Visibility <- "pump_run"
   GraphicView "Template_Graphic view_18" at 509,241 size 88x50; Picture "Graphic_18"
      Visibility <- "pump_run"
   GraphicView "Template_Graphic view_19" at 301,239 size 179x50; Picture "Graphic_18"
      Visibility <- "pump_run"
   GraphicView "Template_Graphic view_20" at 645,241 size 30x50; Picture "Graphic_18"
      Visibility <- "pump_run"
   GraphicView "Graphic view_29" at 265,287 size 35x159; Picture "Graphic_21"
      Visibility <- "pump_run"
   GraphicView "Graphic view_30" at 265,238 size 37x52; Picture "Graphic_34"
      Visibility <- "pump_run"
   IOField "I/O field_1" at 398,197 size 66x38; FormatPattern s99.99
      ProcessValue <- "Tag_9"
   IOField "I/O field_2" at 508,198 size 69x38; FormatPattern s99.99
      ProcessValue <- "P4"
   TextField "Text field_1" at 221,447 size 30x20; Text 'bar'
   GraphicView "Template_Graphic view_22" at 306,483 size 400x65; Picture "Graphic_18"
      Visibility <- "pump_run"
   GraphicView "Template_Graphic view_23" at 735,483 size 98x65; Picture "Graphic_18"
      Visibility <- "pump_run"
   GraphicView "Template_Graphic view_7" at 579,417 size 68x123; Picture "Graphic_15"
   GraphicView "Graphic view_31" at 831,483 size 49x65; Picture "Graphic_33"
      Visibility <- "pump_run"
   GraphicView "Graphic view_32" at 834,354 size 49x108; Picture "Graphic_21"
      Visibility <- "pump_run"
   Button "Button_10" at 279,696 size 156x56; TextOn 'Home'; TextOff 'NPSH test'
      on Press: ActivateScreen("NPSH test", 0)
   Button "Button_11" at 32,694 size 220x56; TextOff 'Performance test'
      on Press: ActivateScreen("performance_1", 0)
   IOField "I/O field_3" at 426,339 size 67x42; FormatPattern 9999
      ProcessValue <- "Referance_motor_speed"
   TextField "Text field_3" at 386,426 size 38x20; Text 'P1'
   TextField "Text field_4" at 223,388 size 38x20; Text 'P2'
   TextField "Text field_2" at 307,334 size 113x48; Text 'Referance speed'
   TextField "Text field_5" at 427,171 size 38x20; Text 'P3'
   TextField "Text field_6" at 534,176 size 38x20; Text 'P4'
   Button "Button_1" at 664,634 size 155x56; TextOff 'Start'
      on Press: SetBit("start_motor")
      Appearance <- "pump_run"
   Button "Button_3" at 665,695 size 156x56; TextOff 'Stop'
      on Press: ResetBit("start_motor")
      Appearance <- "pump_run"
   Button "Button_4" at 578,381 size 70x36; TextOff 'Open'
      on Press: function_b14e0dd5("stepp1_start", 0)
      Appearance <- "stepp1_start"
   IOField "I/O field_4" at 581,341 size 64x32; FormatPattern 999
      ProcessValue <- "stepp1_distance"
   IOField "I/O field_5" at 227,571 size 68x32; FormatPattern 999.9; Unit   C
      ProcessValue <- "Temperature"
   Button "Button_5" at 589,154 size 70x36; TextOff 'Open'
      on Press: function_b14e0dd5("stepp2_excut", 0)
      Appearance <- "stepp2_excut"
   IOField "I/O field_6" at 590,113 size 64x32; FormatPattern 999
      ProcessValue <- "stepp2_distance"
   Button "Button_6" at 922,67 size 92x40; TextOff 'Stepp1_Enab.'
      on Press: InvertBit("stepp1_enab")
      Appearance <- "stepp1_enab"
   Button "Button_7" at 921,111 size 94x38; TextOff 'Stepp1_Home.'
      on Press: function_b14e0dd5("stepp1_home", 0)
      Appearance <- "stepp1_home"
   Button "Button_8" at 921,172 size 94x38; TextOff 'Stepp2_Enab.'
      on Press: InvertBit("stepp2_enab")
      Appearance <- "stepp2_enab"
   Button "Button_9" at 922,217 size 94x37; TextOff 'Stepp2_Home.'
      on Press: function_b14e0dd5("stepp2_home", 0)
      Appearance <- "stepp2_home"
   IOField "I/O field_8" at 390,16 size 105x32; FormatPattern 99999999999999999999
      ProcessValue <- "date"
   IOField "I/O field_9" at 612,14 size 107x32; FormatPattern s9999999999
      ProcessValue <- "time"
   TextField "Text field_8" at 40,14 size 157x38; Text 'Impeller configuration'
   TextField "Text field_9" at 526,11 size 81x38; Text 'Start Time'
   TextField "Text field_10" at 334,16 size 66x38; Text 'Date'
   IOField "I/O field_10" at 836,14 size 107x33; FormatPattern s9999999999
      ProcessValue <- "time_1"
   TextField "Text field_11" at 746,9 size 74x38; Text 'End Time'
   IOField "I/O field_11" at 26,330 size 59x57; FormatPattern 99.99
      ProcessValue <- "QARS"
   IOField "I/O field_12" at 86,331 size 59x57; FormatPattern 99.99
      ProcessValue <- "H_ARS"
   IOField "I/O field_13" at 145,331 size 59x57; FormatPattern 9999.9
      ProcessValue <- "SP_ARS"
   TextField "Text field_27" at 147,295 size 52x30; Text 'P.ref'
   TextField "Text field_28" at 159,310 size 27x33; Text 'W'
   TextField "Text field_29" at 28,294 size 58x33; Text 'Q ref'
   TextField "Text field_30" at 39,309 size 43x33; Text 'm3/h'
   TextField "Text field_31" at 87,295 size 54x33; Text 'H ref'
   TextField "Text field_32" at 100,309 size 27x33; Text 'm'
   TextField "Text field_7" at 111,575 size 109x23; Text 'Tempreture'
   IOField "I/O field_7" at 209,18 size 106x31; FormatPattern ?????????
      ProcessValue <- "configuration"
   Button "Button_12" at 459,695 size 190x55; TextOff 'Temp&Vib_trends'
      on Click: ActivateScreen("Temp&Vib_trends", 0)
      on Press: ActivateScreen("Temp&Vib_trends", 0)
   IOField "I/O field_14" at 28,171 size 59x47; FormatPattern 99.99
      ProcessValue <- "Q"
   IOField "I/O field_83" at 85,171 size 59x47; FormatPattern 99.99
      ProcessValue <- "H"
   IOField "I/O field_84" at 143,171 size 59x47; FormatPattern 9999.99
      ProcessValue <- "Shaft_power"
   TextField "Text field_13" at 41,126 size 38x23; Text 'Q'
   TextField "Text field_16" at 43,149 size 42x23; Text 'm3/h'
   TextField "Text field_17" at 97,129 size 33x23; Text 'H'
   TextField "Text field_18" at 102,151 size 24x23; Text 'm'
   TextField "Text field_19" at 137,124 size 63x29; Text 'Shaft p.'
   TextField "Text field_20" at 155,148 size 27x23; Text 'W'
   Button "Button_13" at 36,254 size 153x39; TextOff 'Reference'
   Button "Button_14" at 37,80 size 153x38; TextOff 'Actual'

